// TIA Portal project "DT_PSA_OPCV" (V19)

(* hardware
DEVICE "S7-1500/ET200MP-Station_1"  S7-1500 station
   slot 0: "Profilschiene_0"  Rack  6ES7 590-1***0-0AA0
   slot 1: "PLC_1"  CPU 1516F-3 PN/DP  6ES7 516-3FN02-0AB0  V2.9
      slot 3: "CPU-Display_1"  6ES7591-1BA00-0AA0
      slot 32768: "PROFINET-Schnittstelle_1"  X1
         slot 32769: "Port_1"  X1 P1
         slot 32770: "Port_2"  X1 P2
      slot 33024: "PROFINET-Schnittstelle_2"  X2
         slot 33025: "Port_1"  X2 P1
      slot 33280: "DP-Schnittstelle_1"  X3
      slot 34817: "Virtual CP interface port_1"  Virtual CP interface port  Virtual CP interface port
   slot 2: "DI 16x24VDC HF_1"  DI 16x24VDC HF  6ES7 521-1BH00-0AB0  V2.2
   slot 3: "DQ 8x24VDC/2A HF_1"  DQ 8x24VDC/2A HF  6ES7 522-1BF00-0AB0  V2.2
   slot 4: "F-DI 16x24V DC_1"  F-DI 16x24V DC  6ES7 526-1BH00-0AB0  V1.0
      slot 1: "F-DI 16x24V DC_1"  F-DI 16x24V DC
   slot 5: "F-DQ 8x24V DC/2A PPM_1"  F-DQ 8x24V DC/2A PPM  6ES7 526-2BF00-0AB0  V1.0
      slot 1: "F-DQ 8x24V DC/2A PPM_1"  F-DQ 8x24V DC/2A PPM
DEVICE "HMI_1"  TP700 Comfort
   slot 0: "HMI_1"  TP700 Comfort  6AV2 124-0GC01-0AX0  17.0.0.0
   slot 1: "HMI_RT_1"  TP700 Comfort  6AV2 124-0GC01-0AX0  17.0.0.0
   slot 5: "HMI_1.IE_CP_1"  PROFINET Interface  17.0.0.0
      slot 1: "PROFINET Schnittstelle_1"  PROFINET Interface
         slot 1: "Port_1"  Port
         slot 2: "Port_2"  Port
   slot 7: "HMI_1.MPI/DP_CP_1"  MPI/DP Interface  17.0.0.0
*)

// ===== PLC "PLC_1"  CPU 1516F-3 PN/DP =====
// protected blocks, not shown: "Main_Safety_RTG1", "Main_Safety_RTG1_DB"

VAR_GLOBAL   // PLC tag table "Control Panel"
   "BT2_OpMode" AT %I0.2 : Bool;   // Betriebsart: 1=Automatik / 0=Hand / Operating mode: 1 = Automatic / 0 = Manual
   "BT3_SingleStep" AT %I0.3 : Bool;   // Einzelschritt ausführen / Execute single step
   "BT4_AutoStart" AT %I0.4 : Bool;   // Automatik Ein / Automatic on
   "BT5_AutoStop" AT %I0.5 : Bool;   // Automatik Halt / Automatic stop
   "BT7_Reset" AT %I0.7 : Bool;   // Grundstellung / Home position
   "BT6_Ack" AT %I0.6 : Bool;   // Störung quittieren / Acknowledge fault
   "BT1_ControlLight" AT %Q0.1 : Bool;   // Tasterbeleuchtung "Steuerung läuft" (grün) / Pushbutton illumination: "Control running" (green)
   "BT4_AutoLight" AT %Q0.4 : Bool;   // Tasterbeleuchtung "Automatik läuft" (grün) / Pushbutton illumination: "Automatic running" (green)
   "BT6_ErrFltLight" AT %Q0.6 : Bool;   // Tasterbeleuchtung "Lampe Störung" (rot) / Pushbutton illumination: "Fault indicator" (red)
   "SignalTower_Yellow" AT %Q1.2 : Bool;   // Ampel "Lampe Einrichten aktiv" (gelb) / Signal tower: "Setup active" (yellow)
   "BT1_ControlOnOff" AT %I0.1 : Bool;   // 1 = Steuerung Ein (einrastend) / 1 = Control on (latching)
   "SignalTower_Green" AT %Q1.1 : Bool;   // Ampel "Automatik läuft" (grün) / Signal tower: "Automatic running" (green)
   "SignalTower_Red" AT %Q1.3 : Bool;   // Ampel "Störung" (rot) / Signal tower: "Fault" (red)
   "BT3_SingleStepLight" AT %Q0.3 : Bool;   // Tasterbeleuchtung "Einzelschritt läuft" (grün) / Pushbutton illumination: "Single step running" (green)
   "BT7_HomingLight" AT %Q0.7 : Bool;   // Tasterbeleuchtung „Grundstellungsfahrt läuft“ (grün) / Pushbutton illumination: "Homing in progress" (green)
   "BT5_AutoStopLight" AT %Q0.5 : Bool;   // Tasterbeleuchtung "Automatikstopp läuft" (blau) / Pushbutton illumination: "Automatic stopping" (blue)
   "BT8_ImmediateStop" AT %I1.0 : Bool;   // Sofort Halt / Immediate stop
   "BT8_ImmediateStopLight" AT %Q1.0 : Bool;   // Tasterbeleuchtung "Sofort Halt" (rot) / Pushbutton illumination: "Immediate stop" (red)
   "SignalTower_Blue" AT %Q1.4 : Bool;   // Ampel "Automatik stoppt" (blau) / Signal tower: "Automatic stopping" (blue)
   "q_SS_ESTOP1" AT %Q0.0 : Bool;   // Beleuchtung Not-Aus 1 / Emergency stop 1 illumination
   "q_SS_ESTOP2" AT %Q0.2 : Bool;   // Beleuchtung Not-Aus 2 / Emergency stop 2 illumination
END_VAR

VAR_GLOBAL   // PLC tag table "System"
   "Clock_Byte" AT %MB0 : Byte;
   "Clock_10Hz" AT %M0.0 : Bool;
   "Clock_5Hz" AT %M0.1 : Bool;
   "Clock_2.5Hz" AT %M0.2 : Bool;
   "Clock_2Hz" AT %M0.3 : Bool;
   "Clock_1.25Hz" AT %M0.4 : Bool;
   "Clock_1Hz" AT %M0.5 : Bool;
   "Clock_0.625Hz" AT %M0.6 : Bool;
   "Clock_0.5Hz" AT %M0.7 : Bool;
   "System_Byte" AT %MB1 : Byte;
   "FirstScan" AT %M1.0 : Bool;
   "DiagStatusUpdate" AT %M1.1 : Bool;
   "AlwaysTRUE" AT %M1.2 : Bool;
   "AlwaysFALSE" AT %M1.3 : Bool;
   "Commissioning_True" AT %M2.0 : Bool;
END_VAR

VAR_GLOBAL CONSTANT   // PLC tag table "System"
   "SYS_MACHINE_MAXSTATIONS" : USInt := 10;   // Anzahl Stationen pro Maschine / Number of stations per machine
   "SYS_SQ_MAXSEQUENCES" : USInt := 12;   // Anzahl Schrittketten pro Station / Number of sequences per station
   "SYS_DRIVE_POSITIONS" : USInt := 8;   // Anzahl Positionen pro Servoantrieb / Number of positions per servo drive
   "SYS_MANUALMOVEMENTS" : UInt := 64;   // Maximale Anzahl an Einrichtfunktionen / Maximum number of setup functions
   "SYS_HMI_SETUPMAXROWS" : USInt := 6;   // HMI-Vorgabe: maximale Anzahl der auf der Steuerung verfügbaren Einrichtzeilen / HMI setting: maximum number of setup rows available on the PLC
   "SYS_CYCLETIMES" : Int := 10;   // Anzahl Zykluszeitauswertungen / Number of cycle time evaluations
END_VAR

VAR_GLOBAL   // PLC tag table "FG01"
   "FG01_Y_Gripper_InHome" AT %I101.0 : Bool;   // geöffnet / open
   "FG01_Y_Gripper_InWork" AT %I101.1 : Bool;   // geschlossen / closed
   "FG01_Y_Gripper_WorkPos" AT %Q101.1 : Bool;   // schließen / close
   "FG01_Y_Plattform_InHome" AT %I102.0 : Bool;   // hinten / rear
   "FG01_Y_Plattform_InWork" AT %I102.1 : Bool;   // vorne / front
   "FG01_Y_Plattform_HomePos" AT %Q102.0 : Bool;
   "FG01_Y_Plattform_WorkPos" AT %Q102.1 : Bool;
   "FG01_Y_ReaderWindow_InWork" AT %I103.1 : Bool;
   "FG01_Y_ReaderWindow_WorkPos" AT %Q103.1 : Bool;   // Position zum Lesen des Codes / Code reading position
   "FG01_Y_Gripper_HomePos" AT %Q101.0 : Bool;   // öffnen / open
   "FG01_Y_ReaderWindow_HomePos" AT %Q103.0 : Bool;
   "FG01_Y_Gate_1_InHome" AT %I104.0 : Bool;   // geöffnet / open
   "FG01_Y_Gate_1_InWork" AT %I104.1 : Bool;   // geschlossen / closed
   "FG01_Y_Gate_1_WorkPos" AT %Q104.1 : Bool;   // Schließen / Close
   "FG01_Y_Gate_2_InHome" AT %I105.0 : Bool;   // geöffnet / open
   "FG01_Y_Gate_2_InWork" AT %I105.1 : Bool;   // geschlossen / closed
   "FG01_Y_Gate_2_WorkPos" AT %Q105.1 : Bool;   // Schließen / Close
   "FG01_Y_LaserMark" AT %Q107.0 : Bool;
   "FG01_P_Camera.bEnable" AT %Q108.0 : Bool;
   "FG01_P_Camera.bTrigger" AT %Q108.1 : Bool;
   "FG01_P_Camera.bReady" AT %I108.0 : Bool;
   "FG01_P_Camera.bBusy" AT %I108.1 : Bool;
   "FG01_P_Camera.bResultValid" AT %I108.2 : Bool;
   "FG01_P_Camera.bResultOk" AT %I108.3 : Bool;
END_VAR

VAR_GLOBAL   // PLC tag table "FG02"
   "FG02_P_Camera.bEnable" AT %Q200.0 : Bool;
   "FG02_P_Camera.bTrigger" AT %Q200.1 : Bool;
   "FG02_P_Camera.bReady" AT %I200.0 : Bool;
   "FG02_P_Camera.bBusy" AT %I200.1 : Bool;
   "FG02_P_Camera.bResultValid" AT %I200.2 : Bool;
   "FG02_P_Camera.bResultOk" AT %I200.3 : Bool;
END_VAR

VAR_GLOBAL   // PLC tag table "FG03"
   "FG03_Y_AxisR1_InHome" AT %I301.0 : Bool;
   "FG03_Y_AxisR1_InWork" AT %I301.1 : Bool;
   "FG03_Y_AxisR1_HomePos" AT %Q301.0 : Bool;
   "FG03_Y_AxisR1_WorkPos" AT %Q301.1 : Bool;
   "FG03_Y_AxisX1_InHome" AT %I302.0 : Bool;
   "FG03_Y_AxisX1_InWork" AT %I302.1 : Bool;
   "FG03_Y_AxisX1_HomePos" AT %Q302.0 : Bool;
   "FG03_Y_AxisX1_WorkPos" AT %Q302.1 : Bool;
   "FG03_Y_AxisY1_InHome" AT %I303.0 : Bool;
   "FG03_Y_AxisY1_InWork" AT %I303.1 : Bool;
   "FG03_Y_AxisY1_HomePos" AT %Q303.0 : Bool;
   "FG03_Y_AxisY1_WorkPos" AT %Q303.1 : Bool;
   "FG03_Y_AxisX2_InHome" AT %I304.0 : Bool;
   "FG03_Y_AxisX2_InWork" AT %I304.1 : Bool;
   "FG03_Y_AxisX2_HomePos" AT %Q304.0 : Bool;
   "FG03_Y_AxisX2_WorkPos" AT %Q304.1 : Bool;
   "FG03_Y_AxisY2_InHome" AT %I305.0 : Bool;
   "FG03_Y_AxisY2_InWork" AT %I305.1 : Bool;
   "FG03_Y_AxisY2_HomePos" AT %Q305.0 : Bool;
   "FG03_Y_AxisY2_WorkPos" AT %Q305.1 : Bool;
   "FG03_Y_Gripper1_InHome" AT %I306.0 : Bool;
   "FG03_Y_Gripper1_InWork" AT %I306.1 : Bool;
   "FG03_Y_Gripper1_HomePos" AT %Q306.0 : Bool;
   "FG03_Y_Gripper1_WorkPos" AT %Q306.1 : Bool;
   "FG03_Y_Gripper2_InHome" AT %I307.0 : Bool;
   "FG03_Y_Gripper2_InWork" AT %I307.1 : Bool;
   "FG03_Y_Gripper2_HomePos" AT %Q307.0 : Bool;
   "FG03_Y_Gripper2_WorkPos" AT %Q307.1 : Bool;
END_VAR

VAR_GLOBAL   // PLC tag table "FG04"
   "FG04_Y_AxisZ_InWork" AT %I401.1 : Bool;
   "FG04_Y_AxisZ_WorkPos" AT %Q401.1 : Bool;
   "FG04_Y_AxisZ_HomePos" AT %Q401.0 : Bool;
   "FG04_Y_AxisZ_InHome" AT %I401.0 : Bool;
END_VAR

VAR_GLOBAL   // PLC tag table "FG05"
   "FG05_B_Part" AT %I500.0 : Bool;
   "FG05_Y_AxisR_InHome" AT %I501.0 : Bool;
   "FG05_Y_AxisR_InWork" AT %I501.1 : Bool;
   "FG05_Y_AxisR_HomePos" AT %Q501.0 : Bool;
   "FG05_Y_AxisR_WorkPos" AT %Q501.1 : Bool;
   "FG05_Y_AxisX_InHome" AT %I502.0 : Bool;
   "FG05_Y_AxisX_InWork" AT %I502.1 : Bool;
   "FG05_Y_AxisX_HomePos" AT %Q502.0 : Bool;
   "FG05_Y_AxisX_WorkPos" AT %Q502.1 : Bool;
   "FG05_Y_AxisZ1_InHome" AT %I503.0 : Bool;
   "FG05_Y_AxisZ1_InWork" AT %I503.1 : Bool;
   "FG05_Y_AxisZ1_HomePos" AT %Q503.0 : Bool;
   "FG05_Y_AxisZ1_WorkPos" AT %Q503.1 : Bool;
   "FG05_Y_AxisZ2_InHome" AT %I504.0 : Bool;
   "FG05_Y_AxisZ2_InWork" AT %I504.1 : Bool;
   "FG05_Y_AxisZ2_HomePos" AT %Q504.0 : Bool;
   "FG05_Y_AxisZ2_WorkPos" AT %Q504.1 : Bool;
   "FG05_Y_CapsSourceStopper_InHome" AT %I505.0 : Bool;   // GS = Kappen können vereinzelt werden / GS = Caps can be separated
   "FG05_Y_CapsSourceStopper_WorkPos" AT %Q505.1 : Bool;   // AS = Vereinzelung kann geleert werden (Vereinzelung nicht möglich) / AS = Separator can be emptied (separation not possible)
   "FG05_Y_Gripper_InHome" AT %I506.0 : Bool;
   "FG05_Y_Gripper_InWork" AT %I506.1 : Bool;
   "FG05_Y_Gripper_HomePos" AT %Q506.0 : Bool;
   "FG05_Y_Gripper_WorkPos" AT %Q506.1 : Bool;
   "FG05_Y_CapsSourceStopper_HomePos" AT %Q505.0 : Bool;
   "FG05_M_Bunker" AT %Q507.0 : Bool;   // Sortiertopf ein / Bowl feeder on
   "FG05_M_Conveyor" AT %Q507.1 : Bool;   // Linearförderer ein / Linear conveyor on
   "FG05_P_Camera.bEnable" AT %Q508.0 : Bool;
   "FG05_P_Camera.bTrigger" AT %Q508.1 : Bool;
   "FG05_P_Camera.bReady" AT %I508.0 : Bool;
   "FG05_P_Camera.bBusy" AT %I508.1 : Bool;
   "FG05_P_Camera.bResultValid" AT %I508.2 : Bool;
   "FG05_P_Camera.bResultOk" AT %I508.3 : Bool;
END_VAR

VAR_GLOBAL   // PLC tag table "FG_Transport"
   "FG_TS_Index01_B_Detect" AT %I1003.0 : Bool;   // 1 = erkannt / 1 = Detected
   "FG_TS_Index01_B_Exit" AT %I1003.1 : Bool;   // 1 = erkannt / 1 = Detected
   "FG_TS_Index01_Y_Lift_InHome" AT %I1003.2 : Bool;   // Heber ist unten / Lift is down
   "FG_TS_Index01_Y_Lift_InWork" AT %I1003.3 : Bool;   // Heber ist oben / Lift is up
   "FG_TS_Index01_Y_Lift_HomePos" AT %Q1003.0 : Bool;   // Heber senken / Lower lift
   "FG_TS_Index01_Y_Lift_WorkPos" AT %Q1003.1 : Bool;   // Heber heben / Raise lift
   "FG_TS_Index01_Y_Stopper_InHome" AT %I1003.4 : Bool;   // Stopper geschlossen / Stopper closed
   "FG_TS_Index01_Y_Stopper_WorkPos" AT %Q1003.2 : Bool;   // Stopper öffnen / Open stopper
   "FG_TS_Index02_B_Detect" AT %I1004.0 : Bool;   // 1 = erkannt / 1 = Detected
   "FG_TS_Index02_B_Exit" AT %I1004.1 : Bool;   // 1 = erkannt / 1 = Detected
   "FG_TS_Index02_Y_Lift_InHome" AT %I1004.2 : Bool;   // Heber ist unten / Lift is down
   "FG_TS_Index02_Y_Lift_InWork" AT %I1004.3 : Bool;   // Heber ist oben / Lift is up
   "FG_TS_Index02_Y_Lift_HomePos" AT %Q1004.0 : Bool;   // Heber senken / Lower lift
   "FG_TS_Index02_Y_Lift_WorkPos" AT %Q1004.1 : Bool;   // Heber heben / Raise lift
   "FG_TS_Index02_Y_Stopper_InHome" AT %I1004.4 : Bool;   // Stopper geschlossen / Stopper closed
   "FG_TS_Index02_Y_Stopper_WorkPos" AT %Q1004.2 : Bool;   // Stopper öffnen / Open stopper
   "FG_TS_Index03_B_Detect" AT %I1005.0 : Bool;   // 1 = erkannt / 1 = Detected
   "FG_TS_Index03_B_Exit" AT %I1005.1 : Bool;   // 1 = erkannt / 1 = Detected
   "FG_TS_Index03_Y_Lift_InHome" AT %I1005.2 : Bool;   // Heber ist unten / Lift is down
   "FG_TS_Index03_Y_Lift_InWork" AT %I1005.3 : Bool;   // Heber ist oben / Lift is up
   "FG_TS_Index03_Y_Lift_HomePos" AT %Q1005.0 : Bool;   // Heber senken / Lower lift
   "FG_TS_Index03_Y_Lift_WorkPos" AT %Q1005.1 : Bool;   // Heber heben / Raise lift
   "FG_TS_Index03_Y_Stopper_InHome" AT %I1005.4 : Bool;   // Stopper geschlossen / Stopper closed
   "FG_TS_Index03_Y_Stopper_WorkPos" AT %Q1005.2 : Bool;   // Stopper öffnen / Open stopper
   "FG_TS_Index04_B_Detect" AT %I1006.0 : Bool;   // 1 = erkannt / 1 = Detected
   "FG_TS_Index04_B_Exit" AT %I1006.1 : Bool;   // 1 = erkannt / 1 = Detected
   "FG_TS_Index04_Y_Lift_InHome" AT %I1006.2 : Bool;   // Heber ist unten / Lift is down
   "FG_TS_Index04_Y_Lift_InWork" AT %I1006.3 : Bool;   // Heber ist oben / Lift is up
   "FG_TS_Index04_Y_Lift_HomePos" AT %Q1006.0 : Bool;   // Heber senken / Lower lift
   "FG_TS_Index04_Y_Lift_WorkPos" AT %Q1006.1 : Bool;   // Heber heben / Raise lift
   "FG_TS_Index04_Y_Stopper_InHome" AT %I1006.4 : Bool;   // Stopper geschlossen / Stopper closed
   "FG_TS_Index04_Y_Stopper_WorkPos" AT %Q1006.2 : Bool;   // Stopper öffnen / Open stopper
   "FG_TS_Index05_B_Detect" AT %I1007.0 : Bool;   // 1 = erkannt / 1 = Detected
   "FG_TS_Index05_B_Exit" AT %I1007.1 : Bool;   // 1 = erkannt / 1 = Detected
   "FG_TS_Index05_Y_Lift_InHome" AT %I1007.2 : Bool;   // Heber ist unten / Lift is down
   "FG_TS_Index05_Y_Lift_InWork" AT %I1007.3 : Bool;   // Heber ist oben / Lift is up
   "FG_TS_Index05_Y_Lift_HomePos" AT %Q1007.0 : Bool;   // Heber senken / Lower lift
   "FG_TS_Index05_Y_Lift_WorkPos" AT %Q1007.1 : Bool;   // Heber heben / Raise lift
   "FG_TS_Index05_Y_Stopper_InHome" AT %I1007.4 : Bool;   // Stopper geschlossen / Stopper closed
   "FG_TS_Index05_Y_Stopper_WorkPos" AT %Q1007.2 : Bool;   // Stopper öffnen / Open stopper
   "FG_TS_Stopper01_B_Detect" AT %I1008.0 : Bool;   // 1 = erkannt / 1 = Detected
   "FG_TS_Stopper01_B_Exit" AT %I1008.1 : Bool;   // 1 = erkannt / 1 = Detected
   "FG_TS_Stopper01_Y_Stopper_InHome" AT %I1008.4 : Bool;   // Stopper geschlossen / Stopper closed
   "FG_TS_Stopper01_Y_Stopper_WorkPos" AT %Q1008.2 : Bool;   // Stopper öffnen / Open stopper
   "FG_TS_Stopper02_B_Detect" AT %I1009.0 : Bool;   // 1 = erkannt / 1 = Detected
   "FG_TS_Stopper02_B_Exit" AT %I1009.1 : Bool;   // 1 = erkannt / 1 = Detected
   "FG_TS_Stopper02_Y_Stopper_InHome" AT %I1009.4 : Bool;   // Stopper geschlossen / Stopper closed
   "FG_TS_Stopper02_Y_Stopper_WorkPos" AT %Q1009.2 : Bool;   // Stopper öffnen / Open stopper
   "FG_TS_Stopper03_B_Detect" AT %I1010.0 : Bool;   // 1 = erkannt / 1 = Detected
   "FG_TS_Stopper03_B_Exit" AT %I1010.1 : Bool;   // 1 = erkannt / 1 = Detected
   "FG_TS_Stopper03_Y_Stopper_InHome" AT %I1010.4 : Bool;   // Stopper geschlossen / Stopper closed
   "FG_TS_Stopper03_Y_Stopper_WorkPos" AT %Q1010.2 : Bool;   // Stopper öffnen / Open stopper
   "FG_TS_Stopper04_B_Detect" AT %I1011.0 : Bool;   // 1 = erkannt / 1 = Detected
   "FG_TS_Stopper04_B_Exit" AT %I1011.1 : Bool;   // 1 = erkannt / 1 = Detected
   "FG_TS_Stopper04_Y_Stopper_InHome" AT %I1011.4 : Bool;   // Stopper geschlossen / Stopper closed
   "FG_TS_Stopper04_Y_Stopper_WorkPos" AT %Q1011.2 : Bool;   // Stopper öffnen / Open stopper
   "FG_TS_Lift01_B_Detect" AT %I1012.0 : Bool;   // 1 = erkannt / 1 = Detected
   "FG_TS_Lift01_B_Exit" AT %I1012.1 : Bool;   // 1 = erkannt / 1 = Detected
   "FG_TS_Lift01_Y_Lift_InHome" AT %I1012.2 : Bool;   // Heber ist unten / Lift is down
   "FG_TS_Lift01_Y_Lift_InWork" AT %I1012.3 : Bool;   // Heber ist oben / Lift is up
   "FG_TS_Lift01_Y_Lift_HomePos" AT %Q1012.0 : Bool;   // Heber senken / Lower lift
   "FG_TS_Lift01_Y_Lift_WorkPos" AT %Q1012.1 : Bool;   // Heber heben / Raise lift
   "FG_TS_Lift01_M_Conveyor_Plus" AT %Q1012.2 : Bool;   // Antrieb vorwärts / Drive forwards
   "FG_TS_Lift01_M_Conveyor_Minus" AT %Q1012.3 : Bool;   // Antrieb rückwärts / Drive backwards
   "FG_TS_Lift02_B_Detect" AT %I1013.0 : Bool;   // 1 = erkannt / 1 = Detected
   "FG_TS_Lift02_B_Exit" AT %I1013.1 : Bool;   // 1 = erkannt / 1 = Detected
   "FG_TS_Lift02_Y_Lift_InHome" AT %I1013.2 : Bool;   // Heber ist unten / Lift is down
   "FG_TS_Lift02_Y_Lift_InWork" AT %I1013.3 : Bool;   // Heber ist oben / Lift is up
   "FG_TS_Lift02_Y_Lift_HomePos" AT %Q1013.0 : Bool;   // Heber senken / Lower lift
   "FG_TS_Lift02_Y_Lift_WorkPos" AT %Q1013.1 : Bool;   // Heber heben / Raise lift
   "FG_TS_Lift02_M_Conveyor_Plus" AT %Q1013.2 : Bool;   // Antrieb vorwärts / Drive forwards
   "FG_TS_Lift02_M_Conveyor_Minus" AT %Q1013.3 : Bool;   // Antrieb rückwärts / Drive backwards
   "FG_TS_Transport01_M_Conveyor_Plus" AT %Q1014.0 : Bool;   // Antrieb vorwärts / Drive forwards
   "FG_TS_Transport01_M_Conveyor_Minus" AT %Q1014.1 : Bool;   // Antrieb rückwärts / Drive backwards
   "FG_TS_Transport02_M_Conveyor_Plus" AT %Q1015.0 : Bool;   // Antrieb vorwärts / Drive forwards
   "FG_TS_Transport02_M_Conveyor_Minus" AT %Q1015.1 : Bool;   // Antrieb rückwärts / Drive backwards
END_VAR

VAR_GLOBAL   // PLC tag table "Safety"
   "i_SS_ESTOP1" AT %I50.0 : Bool;
   "i_SS_ESTOP2" AT %I50.1 : Bool;
END_VAR

// folder: Actors/ActorTypes

TYPE "typeActor"
   STRUCT
      setHomePos : Bool;   // Grundstellung ansteuern / Command home position
      setWorkPos : Bool;   // Arbeitsstellung ansteuern / Command working position
      inHomePos : Bool;   // steht in Grundstellung / in home position
      inWorkPos : Bool;   // steht in Arbeitsstellung / in working position
      homeAct : Bool;   // Grundstellung wird angesteuert / Home position commanded
      workAct : Bool;   // Arbeitsstellung wird angesteuert / Working position commanded
      homeIsInterlocked : Bool;   // 1 = Grundstellung ist gesperrt / 1 = Home position movement inhibited
      workIsInterlocked : Bool;   // 1 = Arbeitsstellung ist gesperrt / 1 = Working position movement inhibited
   END_STRUCT;
END_TYPE

TYPE "typeActor_2Out0In"
   STRUCT
      setHomePos : Bool;   // Grundstellung ansteuern / Command home position
      setWorkPos : Bool;   // Arbeitsstellung ansteuern / Command working position
      homeAct : Bool;   // Grundstellung wird angesteuert / Home position commanded
      workAct : Bool;   // Arbeitsstellung wird angesteuert / Working position commanded
      homeIsInterlocked : Bool;   // 1 = Grundstellung ist gesperrt / 1 = Home position movement inhibited
      workIsInterlocked : Bool;   // 1 = Arbeitsstellung ist gesperrt / 1 = Working position movement inhibited
      setError : Bool;   // in Störung setzen / Set fault state
      inError : Bool;   // Störung vorhanden / Fault present
   END_STRUCT;
END_TYPE

TYPE "typeActor_2Out2In"
   STRUCT
      setHomePos : Bool;   // Grundstellung ansteuern / Command home position
      setWorkPos : Bool;   // Arbeitsstellung ansteuern / Command working position
      inHomePos : Bool;   // steht in Grundstellung / in home position
      inWorkPos : Bool;   // steht in Arbeitsstellung / in working position
      homeAct : Bool;   // Grundstellung wird angesteuert / Home position commanded
      workAct : Bool;   // Arbeitsstellung wird angesteuert / Working position commanded
      homeIsInterlocked : Bool;   // 1 = Grundstellung ist gesperrt / 1 = Home position movement inhibited
      workIsInterlocked : Bool;   // 1 = Arbeitsstellung ist gesperrt / 1 = Working position movement inhibited
      setError : Bool;   // in Störung setzen / Set fault state
      inError : Bool;   // Störung vorhanden / Fault present
   END_STRUCT;
END_TYPE

TYPE "typeActor_1Out0In"
   STRUCT
      setWorkPos : Bool;   // Arbeitsstellung ansteuern / Command working position
      workAct : Bool;   // Arbeitsstellung wird angesteuert / Working position commanded
      workIsInterlocked : Bool;   // 1 = Arbeitsstellung ist gesperrt / 1 = Working position movement inhibited
      setError : Bool;   // in Störung setzen / Set fault state
      inError : Bool;   // Störung vorhanden / Fault present
   END_STRUCT;
END_TYPE

TYPE "typeActor_1Out2In"
   STRUCT
      setWorkPos : Bool;   // Arbeitsstellung ansteuern / Command working position
      inHomePos : Bool;   // steht in Grundstellung / in home position
      inWorkPos : Bool;   // steht in Arbeitsstellung / in working position
      workAct : Bool;   // Arbeitsstellung wird angesteuert / Working position commanded
      workIsInterlocked : Bool;   // 1 = Arbeitsstellung ist gesperrt / 1 = Working position movement inhibited
      setError : Bool;   // in Störung setzen / Set fault state
      inError : Bool;   // Störung vorhanden / Fault present
   END_STRUCT;
END_TYPE

TYPE "typeActor_2Out1In"
   STRUCT
      setHomePos : Bool;   // Grundstellung ansteuern / Command home position
      setWorkPos : Bool;   // Arbeitsstellung ansteuern / Command working position
      inHomePos : Bool;   // steht in Grundstellung / in home position
      inWorkPos : Bool;   // steht in Arbeitsstellung / in working position
      homeAct : Bool;   // Grundstellung wird angesteuert / Home position commanded
      workAct : Bool;   // Arbeitsstellung wird angesteuert / Working position commanded
      homeIsInterlocked : Bool;   // 1 = Grundstellung ist gesperrt / 1 = Home position movement inhibited
      workIsInterlocked : Bool;   // 1 = Arbeitsstellung ist gesperrt / 1 = Working position movement inhibited
      setError : Bool;   // in Störung setzen / Set fault state
      inError : Bool;   // Störung vorhanden / Fault present
   END_STRUCT;
END_TYPE

TYPE "typeActor_1Out1In"
   STRUCT
      setWorkPos : Bool;   // Arbeitsstellung ansteuern / Command working position
      inHomePos : Bool;   // steht in Grundstellung / in home position
      inWorkPos : Bool;   // steht in Arbeitsstellung / in working position
      workAct : Bool;   // Arbeitsstellung wird angesteuert / Working position commanded
      workIsInterlocked : Bool;   // 1 = Arbeitsstellung ist gesperrt / 1 = Working position movement inhibited
      setError : Bool;   // in Störung setzen / Set fault state
      inError : Bool;   // Störung vorhanden / Fault present
   END_STRUCT;
END_TYPE

TYPE "typeActor_1Out_SimpleCamera"
   STRUCT
      setTrigger : Bool;   // Kamera auslösen / Trigger camera
      isReady : Bool;   // ist bereit / ready
      isBusy : Bool;   // ist aktiv / active
      resultOk : Bool;   // Ergebnis ist IO / Result OK
      resultNok : Bool;   // Ergebnis ist NIO / Result NOK
      triggerAct : Bool;   // Trigger wird angesteuert / Trigger commanded
      workIsInterlocked : Bool;   // Triggern ist gesperrt / Triggering inhibited
      setError : Bool;   // in Störung setzen / Set fault state
      inError : Bool;   // Störung vorhanden / Fault present
   END_STRUCT;
END_TYPE

// folder: Actors/Drives

TYPE "typeDriveData"
   STRUCT
      position : Array[1.."SYS_DRIVE_POSITIONS"] of Real;   // Positionsvorgabe / Position setpoint
      speed : Array[1.."SYS_DRIVE_POSITIONS"] of Real;   // Geschwindigkeitsvorgabe / Speed setpoint
   END_STRUCT;
   // // position[1] : Grundstellung (reserviert) / Home position (reserved)
END_TYPE

TYPE "typeDriveControl"
   STRUCT
      moveToPos : Array[1.."SYS_DRIVE_POSITIONS"] of Bool;   // Fahrbefehl ausführen / Execute motion command
      jog : Struct   // Handbetrieb / Manual operation
         pos : Bool;   // Tippen positiv / Jog positive
         neg : Bool;   // Tippen negativ / Jog negative
         "step" : Real;   // Tippschrittweite / Jog increment
         speed : Real;   // Tippgeschwindigkeit / Jog speed
      END_STRUCT;
   END_STRUCT;
END_TYPE

TYPE "typeDriveStatus"
   STRUCT
      ready : Bool;   // Bereit / Ready
      error : Bool;   // Störung / Fault
      posReached : Bool;   // Positionsvorgabe erreicht / Position setpoint reached
      actualPosition : Real;   // Ist-Position / Actual position
      actualSpeed : Real;   // Ist-Geschwindigkeit / Actual speed
      interlockMin : Bool;   // 1 = Fahrtrichtung zur Endposition min gesperrt / 1 = Movement towards minimum end position inhibited
      interlockMax : Bool;   // 1 = Fahrtrichtung zur Endposition max gesperrt / 1 = Movement towards maximum end position inhibited
      endPosMin : Bool;   // Endposition min erreicht / Minimum end position reached
      endPosMax : Bool;   // Endposition max erreicht / Maximum end position reached
      inHomePos : Bool;   // steht in Grundstellung / in home position
   END_STRUCT;
END_TYPE

TYPE "typeDriveConverter"
   STRUCT
      actualPosition : Real;   // Ist-Position (Antriebseinheit) / Actual position (drive units)
      actualSpeed : Real;   // Ist-Geschwindigkeit (Antriebseinheit) / Actual speed (drive units)
      setPosition : Real;   // Sollposition (Antriebseinheit) / Target position (drive units)
      setSpeed : Real;   // Sollgeschwindigkeit (Antriebseinheit) / Target speed (drive units)
      minPosDrive : Real;   // Minimale Positionierung (Antriebseinheit) / Minimum positioning value (drive units)
      maxPosDrive : Real;   // Maximale Positionierung (Antriebseinheit) / Maximum positioning value (drive units)
      maxSpeedDrive : Real;   // Maximale Geschwindigkeit (Antriebseinheit) / Maximum speed (drive units)
      posOffset : Real;   // Offset für Positionsfensterfreigabe (Antriebseinheit) / Offset for position window enable (drive units)
      ready : Bool;   // Umrichter Bereit / Converter ready
      error : Bool;   // Umrichter Störung / Converter fault
      posReached : Bool;   // Position erreicht / Position reached
      releaseMotion : Bool;   // Bewegungsfreigabe / Movement enable
   END_STRUCT;
END_TYPE

// folder: HMI/Errors_Messages

TYPE "typePlcErrors"
   STRUCT
      errorNo : Array[1..64] of Bool;
   END_STRUCT;
END_TYPE

TYPE "typeHmiErrMsg"
   STRUCT
      message : Array[1..2] of Word;   // Meldung auslösen / Trigger message
      alarmAckPlc : Array[1..8] of Word;   // Fehler auslösen und Quittierung über SPS / Trigger fault and acknowledge via PLC
      ackHmi : Array[1..4] of Word;   // Quittierung über HMI / Acknowledge via HMI
   END_STRUCT;
END_TYPE

TYPE "typePlcErrMsg"
   STRUCT
      messages : "typePlcMessages";
      alarms : "typePlcErrors";
   END_STRUCT;
END_TYPE

TYPE "typePlcMessages"
   STRUCT
      msgNo : Array[1..32] of Bool;
   END_STRUCT;
END_TYPE

// folder: HMI/ManualMovement

TYPE "typeHmiManualMove"
   STRUCT
      move : "typeManualMove";   // Bewegung / Movement
      movementNo : USInt;   // Nummer der Bewegungsfunktion / Movement function number
      textlistFunctionName : UInt;   // Funktionsname: Wert für Textliste / Function name: text list value
      textlistFunctionExecuteLeft : UInt;   // Bewegung Links: Wert für Textliste / Left movement: text list value
      textlistFunctionFinalPosLeft : UInt;   // Endposition Links: Wert für Textliste / Left end position: text list value
      textlistFunctionExecuteRight : UInt;   // Bewegung Rechts: Wert für Textliste / Right movement: text list value
      textlistFunctionFinalPosRight : UInt;   // Endposition Rechts: Wert für Textliste / Right end position: text list value
   END_STRUCT;
END_TYPE

TYPE "typeHmiManualMovement"
   STRUCT
      selection : Struct
         station : USInt;   // Angewählte Station / Selected station
         page : USInt;   // Aktuelle Seite / Current page
         ofMaxPages : USInt;   // von insgesamt verfügbaren Seiten / of total pages
         nextPage : Bool;   // Schaltfläche: Nächste Seite / Button: Next page
         previousPage : Bool;   // Schaltfläche: Vorherige Seite / Button: Previous page
         showSymbols : Bool;   // Schaltfläche: Zeige symbolische Ansicht / Button: Show symbolic view
      END_STRUCT;
      rows : Array[1.."SYS_HMI_SETUPMAXROWS"] of "typeHmiManualMove";
   END_STRUCT;
END_TYPE

// folder: Machine

TYPE "typeMachine"
   STRUCT
      EStopOk : Bool;   // Not-Aus-Kreis ist geschlossen / Emergency stop circuit closed
      RunUpIsActive : Bool;   // Maschinenanlauf aktiv (Hauptluft einschalten, externe Geräte und Hardware hochfahren) / Machine startup active (switch on main air, start external devices and hardware)
      controlOn : Bool;   // Maschinensteuerung ist eingeschaltet / Machine control switched on
      automaticMode : Bool;   // Betriebsart Automatik ist aktiv / Automatic operating mode active
      automaticIsRunning : Bool;   // Automatik (bzw. ReleaseCycle) läuft in mindestens einer Station / Automatic operation (or ReleaseCycle) running in at least one station
      automaticStart : Bool;   // Automatikstart auslösen / Initiate automatic start
      automaticStops : Bool;   // Automatik stoppt / Automatic stopping
      singleStepPulse : Bool;   // Einzelschritt / Single step
      immediateStop : Bool;   // Sofort Halt der Stationen auslösen / Initiate immediate stop of stations
      acknowledge : Bool;   // Quittierung / Acknowledgement
      reset : Bool;   // Neustart/Grundstellung auslösen / Initiate restart/homing
      isInHoldReached : Bool;   // Alle Stationen haben den Haltepunkt erreicht / All stations have reached the stop point
      isInError : Bool;   // Störung vorhanden / Fault present
      isHoming : Bool;   // Maschinengrundstellungsfahrt wird ausgeführt / Machine homing in progress
      isInHome : Bool;   // Alle Stationen sind in Grundstellung / All stations in home position
   END_STRUCT;
END_TYPE

TYPE "typeStation"
   STRUCT
      xExists : Bool := false;   // true = Station existiert / false = Platzhalter / true = Station exists / false = Placeholder
      usiState : USInt;   // 0 = Bearbeitung, 1 = Störung, 2 = Leerlauf, 3 = Nicht in Produktion, 4 = Warten auf Bediener, 5 = Blockiert, 6 = Materialmangel / 0 = Processing, 1 = Fault, 2 = Idle, 3 = Not in production, 4 = Waiting for operator, 5 = Blocked, 6 = Starved
      udtCycleTime : "typeCycleTime";
      udtSignals : "typeStationSignals";
      udtStepSeqs : "typeStepSequences";
   END_STRUCT;
END_TYPE

TYPE "typeStations"
   STRUCT
      station : Array[1.."SYS_MACHINE_MAXSTATIONS"] of "typeStation";
   END_STRUCT;
END_TYPE

TYPE "typeStepSequence"
   STRUCT
      exists : Bool;   // Schrittkette verfügbar / Sequence available
      start : Bool;   // Start Schrittkette / Start sequence
      running : Bool;   // Schrittkette läuft / Sequence running
      done : Bool;   // Schrittkette ist fertig / Sequence complete
      error : Bool;   // Störung vorhanden / Fault present
      init : Bool;   // Initialschritt aktiv / Initial step active
      inHome : Bool;   // Steht in Grundstellung / In home position
      isWaiting : Bool;   // Steht im Warteschritt / Waiting step active
      inHoming : Bool;   // Grundstellungsfahrt aktiv / Homing active
      jogDone : Bool;   // Halbautomatische Weiterschaltung abgeschlossen / Semi-automatic step advance complete
   END_STRUCT;
END_TYPE

TYPE "typeStepSequences"
   STRUCT
      stepSeq : Array[1.."SYS_SQ_MAXSEQUENCES"] of "typeStepSequence";   // Schrittkette / Sequence
   END_STRUCT;
END_TYPE

TYPE "typeMachineSafety"
   STRUCT
      EStopReq : Bool;   // Not-Aus-Kreis Quittierung erforderlich / Emergency stop circuit acknowledgement required
      EStopOk : Bool;   // Not-Aus-Kreis ok / Emergency stop circuit OK
      RunUp : Bool;   // Hochlaufphase (Starte Belüftung der Hauptventilstation) / Startup phase (start pressurising main valve manifold)
      RunUpIsOk : Bool;   // Sicherheitssteuerung ist hochgefahren (Hauptluftversorgung vorhanden, etc) / Safety control started up (main air supply available, etc.)
      Error : Bool;   // Fehler in der Sicherheitssteuerung / Safety control fault
   END_STRUCT;
END_TYPE

TYPE "typeStationSignals"
   STRUCT
      controlOn : Bool;   // Steuerung eingeschaltet / Control switched on
      automaticMode : Bool;   // Automatikmodus angewählt / Automatic mode selected
      modeSetup : Bool;   // Handmodus angewählt / Manual mode selected
      modeAuto : Bool;   // Betriebsart: Automatik aktiv / Operating mode: Automatic active
      modeTap : Bool;   // Betriebsart: Einzelschritt aktiv / Operating mode: Single step active
      releaseCycle : Bool;   // Bearbeitungsfreigabe / Processing enable
      releaseNextJog : Bool;   // Freigabe Weiterschaltung (Zünd-Impuls für Schrittketten) / Step advance enable (trigger pulse for sequences)
      resetCycle : Bool;   // Ablauf neu starten / Restart sequence
      setupActive : Bool;   // Handmodus/Einrichten aktiv (mindestens 1 Aktor ist in Hand bewegt worden) / Manual/setup mode active (at least one actuator moved manually)
      ack : Bool;   // Quittieren / Acknowledge
      singlePulse : Bool;   // Einzelschritt auslösen / Trigger single step
      safetyIsClosed : Bool;   // Sicherheitskreis ist geschlossen / Safety circuit closed
      safetyIsOk : Bool;   // Sicherheitskreis ist geschlossen und verriegelt / Safety circuit closed and locked
      isInAutoStoping : Bool;   // Automatikstopp/Zyklusende angewählt / Automatic stop / end of cycle selected
      isInHoldReached : Bool;   // Haltepunkt wurde erreicht (z. B. Freigabe zum Öffnen des Sicherheitskreises) / Stop point reached (e.g. permission to open safety circuit)
      isStopped : Bool;   // Automatikabläufe/Graphen sind angehalten / Automatic sequences / GRAPH sequences stopped
      isHoming : Bool;   // Grundstellungsablauf aktiv / Homing sequence active
      isInHome : Bool;   // steht in Grundstellung / in home position
      isInError : Bool;   // Störung vorhanden / Fault present
      actorError : Bool;   // Mindestens ein Stationsaktor hat eine Störung (wird in Aktor-Bausteinen gesetzt) / At least one station actuator has a fault (set in actuator blocks)
      internError : Bool;   // Interner Fehler im Framework vorhanden / Internal framework fault present
   END_STRUCT;
END_TYPE

// folder: Machine/Diag

TYPE "typeCycleTime2"
   STRUCT
      xExists : Bool;   // Zykluszeitauswertung vorhanden / Cycle time evaluation available
      xBottleneck : Bool;   // Bei "true" wird dieser Messbereich zur Diagnose der Engpassstelle ausgewertet / If "true", this measurement area is evaluated for bottleneck diagnosis
      xNewCycle : Bool;   // Ein neuer Messwert liegt vor / New measured value available
      udtHmi : "typeCycleTimeHmi";
      stCurrentCycle : Struct   // Aktueller Zyklus / Current cycle
         tActive : Time;   // Aktive Zeit / Active time
         tInHold : Time;   // Angehaltene Zeit / Stopped time
         tOverall : Time;   // Gesamt / Total
      END_STRUCT;
      stLastCycle : Struct   // Letzter Zyklus / Last cycle
         tActive : Time;   // Aktive Zeit / Active time
         tInHold : Time;   // Angehaltene Zeit / Stopped time
         tOverall : Time;   // Gesamt / Total
      END_STRUCT;
   END_STRUCT;
END_TYPE

TYPE "typeCycleTimes2"
   STRUCT
      cycleTime : Array[1.."SYS_CYCLETIMES"] of "typeCycleTime2";
   END_STRUCT;
END_TYPE

TYPE "typeCycleTimeHmi"
   STRUCT
      rSetpointSeconds : Real := 0.0;   // Sollzeit in Sekunden; Werte kleiner oder gleich 0 deaktivieren die Prüfung / Target time in seconds; values less than or equal to 0 disable the check
      rActiveTimeSeconds : Real;   // Letzte abgeschlossene aktive Zykluszeit in Sekunden / Last completed active cycle time in seconds
      xExceeded : Bool;   // TRUE: Letzte aktive Zykluszeit überschreitet die Sollzeit / TRUE: Last active cycle time exceeds target time
   END_STRUCT;
END_TYPE

TYPE "typeCycleTime"
   STRUCT
      xExists : Bool;   // Zykluszeitauswertung vorhanden / Cycle time evaluation available
      xBottleneck : Bool;   // Bei "true" wird dieser Messbereich zur Diagnose der Engpassstelle ausgewertet / If "true", this measurement area is evaluated for bottleneck diagnosis
      xNewCycle : Bool;   // Ein neuer Messwert liegt vor / New measured value available
      udtHmi : "typeCycleTimeHmi";
      stCurrentCycle : Struct   // Aktueller Zyklus / Current cycle
         tState : Array[0..6] of Time;   // Aktive Zeiten in ms je Stationszustand / Active times in ms per station state
         tOverall : Time;   // Gesamtzeit in ms / Total time in ms
      END_STRUCT;
      stLastCycle : Struct   // Letzter Zyklus / Last cycle
         tState : Array[0..6] of Time;   // Aktive Zeiten in ms je Stationszustand / Active times in ms per station state
         tOverall : Time;   // Gesamtzeit in ms / Total time in ms
      END_STRUCT;
   END_STRUCT;
   // // stCurrentCycle.tState[0] : BEARBEITUNG / PROCESSING
   // // stCurrentCycle.tState[1] : STÖRUNG / FAULT
   // // stCurrentCycle.tState[2] : LEERLAUF / IDLE
   // // stCurrentCycle.tState[3] : NICHT IN PRODUKTION / NOT IN PRODUCTION
   // // stCurrentCycle.tState[4] : WARTEN AUF BEDIENER / WAITING FOR OPERATOR
   // // stCurrentCycle.tState[5] : BLOCKIERT / BLOCKED
   // // stCurrentCycle.tState[6] : MATERIALMANGEL / STARVED
   // // stLastCycle.tState[0] : BEARBEITUNG / PROCESSING
   // // stLastCycle.tState[1] : STÖRUNG / FAULT
   // // stLastCycle.tState[2] : LEERLAUF / IDLE
   // // stLastCycle.tState[3] : NICHT IN PRODUKTION / NOT IN PRODUCTION
   // // stLastCycle.tState[4] : WARTEN AUF BEDIENER / WAITING FOR OPERATOR
   // // stLastCycle.tState[5] : BLOCKIERT / BLOCKED
   // // stLastCycle.tState[6] : MATERIALMANGEL / STARVED
END_TYPE

// folder: Machine/ManualMovement

TYPE "typeManualMove"
   STRUCT
      control : "typeManualMoveControl";   // Steuerung / Control
      attributes : "typeManualMoveAttributes";   // Eigenschaften / Properties
   END_STRUCT;
END_TYPE

TYPE "typeManualMoveSetup"
   STRUCT
      initialisation : Struct   // Für den Initialisierungsdurchlauf notwendig / Required for initialisation pass
         execute : Bool;   // Initialisierung der Bewegungsfunktionen ausführen / Execute movement function initialisation
         isActive : Bool;   // Initialisierung läuft / Initialisation in progress
         isDone : Bool;   // Initialisierung abgeschlossen / Initialisation complete
         error : Bool;   // Initialisierung fehlerhaft / Initialisation failed
         currentStationNo : USInt;   // Hilfsspeicher für die Station / Temporary storage for station
         currentMoveNo : USInt;   // Hilfsspeicher für die Bewegungsnummer innerhalb der Station / Temporary storage for movement number within station
         moveNo : USInt;   // Hilfsspeicher für die Bewegungsnummer (maximale Anzahl Stationen wenn initialisiert) / Temporary movement number storage (maximum station count when initialised)
      END_STRUCT;
   END_STRUCT;
END_TYPE

TYPE "typeManualMovements"
   STRUCT
      setup : "typeManualMoveSetup";
      movements : Array[0.."SYS_MANUALMOVEMENTS"] of "typeManualMove";
   END_STRUCT;
   // // movements[0] : Nicht verwendbar / Not usable
END_TYPE

TYPE "typeManualMoveControl"
   STRUCT
      moveHomePos : Bool;   // Grundstellung ansteuern / Command home position
      moveWorkPos : Bool;   // Arbeitsstellung ansteuern / Command working position
      inHomePos : Bool;   // steht in Grundstellung / in home position
      inWorkPos : Bool;   // steht in Arbeitsstellung / in working position
      homeAct : Bool;   // Grundstellung wird angesteuert / Home position commanded
      workAct : Bool;   // Arbeitsstellung wird angesteuert / Working position commanded
      homeIsInterlocked : Bool;   // 1 = Grundstellung ist gesperrt / 1 = Home position movement inhibited
      workIsInterlocked : Bool;   // 1 = Arbeitsstellung ist gesperrt / 1 = Working position movement inhibited
      value : Real;   // Dezimalanzeige / Decimal display
   END_STRUCT;
END_TYPE

TYPE "typeManualMoveAttributes"
   STRUCT
      initialised : Bool;   // Ist initialisiert / Initialised
      showValue : Bool;   // Zeige Dezimalanzeige / Show decimal display
      showName : Bool;   // Zeige Benennung der Einrichtzeile / Show setup row label
      showRecRight : Bool;   // Rechteck rechts anzeigen / Show right rectangle
      showRecLeft : Bool;   // Rechteck links anzeigen / Show left rectangle
      isExecutableRight : Bool;   // Ist ausführbar rechte Seite / Right side executable
      isExecutableLeft : Bool;   // Ist ausführbar linke Seite / Left side executable
      hasEndPositionRight : Bool;   // Zeige Endposition rechte Seite / Display right end position
      hasEndPositionLeft : Bool;   // Zeige Endposition linke Seite / Display left end position
      stationNo : USInt;   // Zugehörige Stationsnummer / Associated station number
      movementNo : USInt;   // Zugehörige Bewegungsnummer innerhalb der Station / Associated movement number within station
   END_STRUCT;
END_TYPE

// folder: 0.Safety - Password:0000

DATA_BLOCK "SafetySignals"   // DB3
{ S7_Optimized_Access := 'TRUE' }
VERSION : 0.1
   VAR
      xEstop1_Ok : Bool;
      xEstop2_Ok : Bool;
      xEstop1_Ack_Req : Bool;
      xEstop2_Ack_Req : Bool;
   END_VAR
BEGIN
END_DATA_BLOCK

// folder: 1. HMI/TP700_HMI_1

DATA_BLOCK "InstHmiManualMovementController"   // DB1003
{ S7_Optimized_Access := 'TRUE' }
VERSION : 0.1
// stored: InstanceOfName HmiManualMovementController
"HmiManualMovementController"
BEGIN
END_DATA_BLOCK

DATA_BLOCK "HmiManualMovement"   // DB1004
{ S7_Optimized_Access := 'TRUE' }
VERSION : 0.1
BEGIN
END_DATA_BLOCK

// folder: 2. Machine

DATA_BLOCK "InstMachine"   // DB1000
{ S7_Optimized_Access := 'TRUE' }
VERSION : 0.1
// stored: InstanceOfName MachineControl
"MachineControl"
BEGIN
END_DATA_BLOCK

DATA_BLOCK "Machine"   // DB1001
{ S7_Optimized_Access := 'TRUE' }
VERSION : 0.1
   VAR
      safety : "typeMachineSafety";
      machine : "typeMachine";
      stations : "typeStations";
   END_VAR
BEGIN
   // stations.station[1] : FG01
   // stations.station[2] : FG02
   // stations.station[3] : FG03
   // stations.station[4] : FG04
   // stations.station[5] : FG05
   // stations.station[6] : Reserve / Spare
   // stations.station[7] : Reserve / Spare
   // stations.station[8] : Reserve / Spare
   // stations.station[9] : Reserve / Spare
   // stations.station[10] : Transport
   // stations.station[10].udtStepSeqs.stepSeq[1] : Stopper01
   // stations.station[10].udtStepSeqs.stepSeq[2] : Stopper02
   // stations.station[10].udtStepSeqs.stepSeq[3] : Lift01
   // stations.station[10].udtStepSeqs.stepSeq[4] : Stopper03
   // stations.station[10].udtStepSeqs.stepSeq[5] : Index01
   // stations.station[10].udtStepSeqs.stepSeq[6] : Index02
   // stations.station[10].udtStepSeqs.stepSeq[7] : Index03
   // stations.station[10].udtStepSeqs.stepSeq[8] : Index04
   // stations.station[10].udtStepSeqs.stepSeq[9] : Index05
   // stations.station[10].udtStepSeqs.stepSeq[10] : Stopper04
   // stations.station[10].udtStepSeqs.stepSeq[11] : Lift 2
END_DATA_BLOCK

DATA_BLOCK "MachineGlobals"   // DB1002
{ S7_Optimized_Access := 'TRUE' }
VERSION : 0.1
   VAR
      emptying : Bool;   // Maschine leerfahren / Empty machine
   END_VAR
BEGIN
END_DATA_BLOCK

DATA_BLOCK "ManualMovements"   // DB1005
{ S7_Optimized_Access := 'TRUE' }
VERSION : 0.1
BEGIN
END_DATA_BLOCK

// folder: 2. Machine/00_Alarms and Messages

DATA_BLOCK "Alarmserver"   // DB2
{ S7_Optimized_Access := 'TRUE' }
VERSION : 0.1
   VAR
      plc : Struct   // Meldungsspeicher für SPS / Message memory for PLC
         machine : "typePlcErrMsg";
         fg_1 : "typePlcErrMsg";
         fg_2 : "typePlcErrMsg";
         fg_3 : "typePlcErrMsg";
         fg_4 : "typePlcErrMsg";
         fg_5 : "typePlcErrMsg";
         fg_transport : "typePlcErrMsg";
      END_STRUCT;
      hmi : Struct   // Meldungsspeicher für HMI / Message memory for HMI
         machine : "typeHmiErrMsg";
         fg_1 : "typeHmiErrMsg";
         fg_2 : "typeHmiErrMsg";
         fg_3 : "typeHmiErrMsg";
         fg_4 : "typeHmiErrMsg";
         fg_5 : "typeHmiErrMsg";
         fg_transport : "typeHmiErrMsg";
      END_STRUCT;
   END_VAR
BEGIN
END_DATA_BLOCK

// folder: 2. Machine/01_FG01

DATA_BLOCK "InstFG01Control"   // DB1100
{ S7_Optimized_Access := 'TRUE' }
VERSION : 0.1
// stored: InstanceOfName FG01Control
"FG01Control"
BEGIN
END_DATA_BLOCK

DATA_BLOCK "FG01Parameter"   // DB1101
{ S7_Optimized_Access := 'TRUE' }
VERSION : 0.1
BEGIN
END_DATA_BLOCK

DATA_BLOCK "FG01Globals"   // DB1102
{ S7_Optimized_Access := 'TRUE' }
VERSION : 0.1
   VAR
      laserOn : Bool := true;   // Laser einschalten / Switch on laser
      SQ1 : Struct
         readyForIndex : Bool;   // Freigabe für den Indexer zum Anheben / Indexer raising enable
         isinHome : Bool;   // Grundstellung vorhanden / Home position reached
      END_STRUCT;
   END_VAR
BEGIN
END_DATA_BLOCK

DATA_BLOCK "FG01Actors"   // DB1103
{ S7_Optimized_Access := 'TRUE' }
VERSION : 0.1
   VAR
      Gripper : "typeActor_2Out2In";   // Greifer / Gripper
      Plattform : "typeActor_2Out2In";   // Laserplattform / Laser platform
      ReaderWindow : "typeActor_2Out1In";   // Laserplattform / Laser platform
      Lasermarker : "typeActor_1Out0In";   // Lasermarkierer / Laser marker
      Gate_1 : "typeActor_1Out2In";   // Seitentor 1 / Side gate 1
      Gate_2 : "typeActor_1Out2In";   // Seitentor 2 / Side gate 2
      Camera : "typeActor_1Out_SimpleCamera";
   END_VAR
BEGIN
END_DATA_BLOCK

// folder: 2. Machine/01_FG01/Stepsequences

DATA_BLOCK "InstSq_1.1"   // DB1111
{ S7_Optimized_Access := 'TRUE' }
VERSION : 0.1
// stored: InstanceOfName Sq_1.1
"Sq_1.1"
BEGIN
END_DATA_BLOCK

// folder: 2. Machine/02_FG02

DATA_BLOCK "InstFG02Control"   // DB1200
{ S7_Optimized_Access := 'TRUE' }
VERSION : 0.1
// stored: InstanceOfName FG02Control
"FG02Control"
BEGIN
END_DATA_BLOCK

DATA_BLOCK "FG02Globals"   // DB1202
{ S7_Optimized_Access := 'TRUE' }
VERSION : 0.1
   VAR
      SQ1 : Struct
         readyForIndex : Bool;   // Freigabe für den Indexer zum Anheben / Indexer raising enable
         isInHome : Bool;   // Grundstellung vorhanden / Home position reached
      END_STRUCT;
   END_VAR
BEGIN
END_DATA_BLOCK

DATA_BLOCK "FG02Actors"   // DB1203
{ S7_Optimized_Access := 'TRUE' }
VERSION : 0.1
   VAR
      P_Camera : "typeActor_1Out_SimpleCamera";
   END_VAR
BEGIN
END_DATA_BLOCK

// folder: 2. Machine/02_FG02/Stepsequences

DATA_BLOCK "InstSq_2.1"   // DB1211
{ S7_Optimized_Access := 'TRUE' }
VERSION : 0.1
// stored: InstanceOfName Sq_2.1
"Sq_2.1"
BEGIN
END_DATA_BLOCK

// folder: 2. Machine/03_FG03

DATA_BLOCK "InstFG03Control"   // DB1300
{ S7_Optimized_Access := 'TRUE' }
VERSION : 0.1
// stored: InstanceOfName FG03Control
"FG03Control"
BEGIN
END_DATA_BLOCK

DATA_BLOCK "FG03Globals"   // DB1302
{ S7_Optimized_Access := 'TRUE' }
VERSION : 0.1
   VAR
      SQ1 : Struct
         readyForIndex : Bool;   // Freigabe für den Indexer zum Anheben / Indexer raising enable
         isInHome : Bool;   // Grundstellung vorhanden / Home position reached
      END_STRUCT;
   END_VAR
BEGIN
END_DATA_BLOCK

DATA_BLOCK "FG03Actors"   // DB1303
{ S7_Optimized_Access := 'TRUE' }
VERSION : 0.1
   VAR
      AxisR1 : "typeActor_2Out2In";
      AxisX1 : "typeActor_2Out2In";
      AxisY1 : "typeActor_2Out2In";
      AxisX2 : "typeActor_2Out2In";
      AxisY2 : "typeActor_2Out2In";
      Gripper1 : "typeActor_2Out2In";
      Gripper2 : "typeActor_2Out2In";
   END_VAR
BEGIN
END_DATA_BLOCK

// folder: 2. Machine/03_FG03/Stepsequences

DATA_BLOCK "InstSq_3.1"   // DB1311
{ S7_Optimized_Access := 'TRUE' }
VERSION : 0.1
// stored: InstanceOfName Sq_3.1
"Sq_3.1"
BEGIN
END_DATA_BLOCK

// folder: 2. Machine/04_FG04

DATA_BLOCK "InstFG04Control"   // DB1400
{ S7_Optimized_Access := 'TRUE' }
VERSION : 0.1
// stored: InstanceOfName FG04Control
"FG04Control"
BEGIN
END_DATA_BLOCK

DATA_BLOCK "FG04Globals"   // DB1402
{ S7_Optimized_Access := 'TRUE' }
VERSION : 0.1
   VAR
      SQ1 : Struct
         readyForIndex : Bool;   // Freigabe für den Indexer zum Anheben / Indexer raising enable
         isInHome : Bool;   // Grundstellung vorhanden / Home position reached
      END_STRUCT;
   END_VAR
BEGIN
END_DATA_BLOCK

DATA_BLOCK "FG04Actors"   // DB1403
{ S7_Optimized_Access := 'TRUE' }
VERSION : 0.1
   VAR
      AxisZ : "typeActor_2Out2In";
   END_VAR
BEGIN
END_DATA_BLOCK

// folder: 2. Machine/04_FG04/Stepsequences

DATA_BLOCK "InstSq_4.1"   // DB1411
{ S7_Optimized_Access := 'TRUE' }
VERSION : 0.1
// stored: InstanceOfName Sq_4.1
"Sq_4.1"
BEGIN
END_DATA_BLOCK

// folder: 2. Machine/05_FG05

DATA_BLOCK "InstFG05Control"   // DB1500
{ S7_Optimized_Access := 'TRUE' }
VERSION : 0.1
// stored: InstanceOfName FG05Control
"FG05Control"
BEGIN
END_DATA_BLOCK

DATA_BLOCK "FG05Globals"   // DB1502
{ S7_Optimized_Access := 'TRUE' }
VERSION : 0.1
   VAR
      emptying : Bool;   // Zuführung leerfahren / Empty infeed
      SQ1 : Struct
         readyForIndex : Bool;   // Freigabe für den Indexer zum Anheben / Indexer raising enable
         isInHome : Bool;   // Grundstellung vorhanden / Home position reached
      END_STRUCT;
   END_VAR
BEGIN
END_DATA_BLOCK

DATA_BLOCK "FG05Actors"   // DB1503
{ S7_Optimized_Access := 'TRUE' }
VERSION : 0.1
   VAR
      AxisR : "typeActor_2Out2In";
      AxisX : "typeActor_2Out2In";
      AxisZ1 : "typeActor_2Out2In";
      AxisZ2 : "typeActor_2Out2In";
      CapsSourceStopper : "typeActor_2Out1In";
      Gripper : "typeActor_2Out2In";
      Bunker : "typeActor_1Out0In";
      Conveyor : "typeActor_1Out0In";
      Camera : "typeActor_1Out_SimpleCamera";
   END_VAR
BEGIN
END_DATA_BLOCK

// folder: 2. Machine/05_FG05/Stepsequences

DATA_BLOCK "InstSq_5.1"   // DB1511
{ S7_Optimized_Access := 'TRUE' }
VERSION : 0.1
// stored: InstanceOfName Sq_5.1
"Sq_5.1"
BEGIN
END_DATA_BLOCK

// folder: 2. Machine/10_FG_Transport

DATA_BLOCK "InstTransportControl"   // DB2000
{ S7_Optimized_Access := 'TRUE' }
VERSION : 0.1
// stored: InstanceOfName TransportControl
"TransportControl"
BEGIN
END_DATA_BLOCK

DATA_BLOCK "TransportGlobals"   // DB2002
{ S7_Optimized_Access := 'TRUE' }
VERSION : 0.1
   VAR
      Index01 : Struct
         release : Bool;   // Startfreigabe für FG01 von Indexer / Start enable for FG01 from indexer
      END_STRUCT;
      Index02 : Struct
         release : Bool;   // Startfreigabe für FG02 von Indexer / Start enable for FG02 from indexer
      END_STRUCT;
      Index03 : Struct
         release : Bool;   // Startfreigabe für FG03 von Indexer / Start enable for FG03 from indexer
      END_STRUCT;
      Index04 : Struct
         release : Bool;   // Startfreigabe für FG04 von Indexer / Start enable for FG04 from indexer
      END_STRUCT;
      Index05 : Struct
         release : Bool;   // Startfreigabe für FG05 von Indexer / Start enable for FG05 from indexer
      END_STRUCT;
   END_VAR
BEGIN
END_DATA_BLOCK

DATA_BLOCK "TransportActors"   // DB2003
{ S7_Optimized_Access := 'TRUE' }
VERSION : 0.1
   VAR
      Index01_Lift : "typeActor_2Out2In";
      Index01_Stopper : "typeActor_1Out1In";
      Index02_Lift : "typeActor_2Out2In";
      Index02_Stopper : "typeActor_1Out1In";
      Index03_Lift : "typeActor_2Out2In";
      Index03_Stopper : "typeActor_1Out1In";
      Index04_Lift : "typeActor_2Out2In";
      Index04_Stopper : "typeActor_1Out1In";
      Index05_Lift : "typeActor_2Out2In";
      Index05_Stopper : "typeActor_1Out1In";
      Stopper01 : "typeActor_1Out1In";
      Stopper02 : "typeActor_1Out1In";
      Stopper03 : "typeActor_1Out1In";
      Stopper04 : "typeActor_1Out1In";
      Lift01_Lift : "typeActor_2Out2In";
      Lift01_Conv : "typeActor_2Out0In";
      Lift02_Lift : "typeActor_2Out2In";
      Lift02_Conv : "typeActor_2Out0In";
      Transport01_Conv : "typeActor_2Out0In";
      Transport02_Conv : "typeActor_2Out0In";
   END_VAR
BEGIN
END_DATA_BLOCK

// folder: 2. Machine/10_FG_Transport/Stepsequences

DATA_BLOCK "InstSq_Stopper01"   // DB2011
{ S7_Optimized_Access := 'TRUE' }
VERSION : 0.1
// stored: InstanceOfName Sq_Process_Stopper
"Sq_Process_Stopper"
BEGIN
END_DATA_BLOCK

DATA_BLOCK "InstSq_Stopper02"   // DB2012
{ S7_Optimized_Access := 'TRUE' }
VERSION : 0.1
// stored: InstanceOfName Sq_Process_Stopper
"Sq_Process_Stopper"
BEGIN
END_DATA_BLOCK

DATA_BLOCK "InstSq_Stopper03"   // DB2013
{ S7_Optimized_Access := 'TRUE' }
VERSION : 0.1
// stored: InstanceOfName Sq_Process_Stopper
"Sq_Process_Stopper"
BEGIN
END_DATA_BLOCK

DATA_BLOCK "InstSq_Stopper04"   // DB2014
{ S7_Optimized_Access := 'TRUE' }
VERSION : 0.1
// stored: InstanceOfName Sq_Process_Stopper
"Sq_Process_Stopper"
BEGIN
END_DATA_BLOCK

DATA_BLOCK "InstSq_Process_Lift1"   // DB2015
{ S7_Optimized_Access := 'TRUE' }
VERSION : 0.1
// stored: InstanceOfName Sq_Process_Lift
"Sq_Process_Lift"
BEGIN
END_DATA_BLOCK

DATA_BLOCK "InstSq_Process_Lift2"   // DB2016
{ S7_Optimized_Access := 'TRUE' }
VERSION : 0.1
// stored: InstanceOfName Sq_Process_Lift
"Sq_Process_Lift"
BEGIN
END_DATA_BLOCK

DATA_BLOCK "InstSq_Process_Index01"   // DB2017
{ S7_Optimized_Access := 'TRUE' }
VERSION : 0.1
// stored: InstanceOfName Sq_Process_IndexingUnit
"Sq_Process_IndexingUnit"
BEGIN
END_DATA_BLOCK

DATA_BLOCK "InstSq_Process_Index02"   // DB2018
{ S7_Optimized_Access := 'TRUE' }
VERSION : 0.1
// stored: InstanceOfName Sq_Process_IndexingUnit
"Sq_Process_IndexingUnit"
BEGIN
END_DATA_BLOCK

DATA_BLOCK "InstSq_Process_Index03"   // DB2019
{ S7_Optimized_Access := 'TRUE' }
VERSION : 0.1
// stored: InstanceOfName Sq_Process_IndexingUnit
"Sq_Process_IndexingUnit"
BEGIN
END_DATA_BLOCK

DATA_BLOCK "InstSq_Process_Index04"   // DB2020
{ S7_Optimized_Access := 'TRUE' }
VERSION : 0.1
// stored: InstanceOfName Sq_Process_IndexingUnit
"Sq_Process_IndexingUnit"
BEGIN
END_DATA_BLOCK

DATA_BLOCK "InstSq_Process_Index05"   // DB2021
{ S7_Optimized_Access := 'TRUE' }
VERSION : 0.1
// stored: InstanceOfName Sq_Process_IndexingUnit
"Sq_Process_IndexingUnit"
BEGIN
END_DATA_BLOCK

DATA_BLOCK "InstTofRunConveyor1"   // DB2030
{ S7_Optimized_Access := 'TRUE' }
AUTHOR : Simatic
FAMILY : IEC
NAME : IEC_TMR
VERSION : 1.0
// stored: InstanceOfName IEC_TIMER
"IEC_TIMER"
BEGIN
END_DATA_BLOCK

DATA_BLOCK "InstTofRunConveyor2"   // DB2031
{ S7_Optimized_Access := 'TRUE' }
AUTHOR : Simatic
FAMILY : IEC
NAME : IEC_TMR
VERSION : 1.0
// stored: InstanceOfName IEC_TIMER
"IEC_TIMER"
BEGIN
END_DATA_BLOCK

// folder: (top level)

ORGANIZATION_BLOCK "Main"   // OB1, LAD, ProgramCycle
TITLE = "Main Program Sweep (Cycle)" / „Zyklischer Hauptprogrammdurchlauf“
{ S7_Optimized_Access := 'TRUE' }
VERSION : 0.1
   VAR_INPUT
      Initial_Call : Bool;   // Initial call of this OB
      Remanence : Bool;   // =True, if remanent data are available
   END_VAR
BEGIN

REGION Network 1: Inbetriebnahme-Merker / Commissioning flag
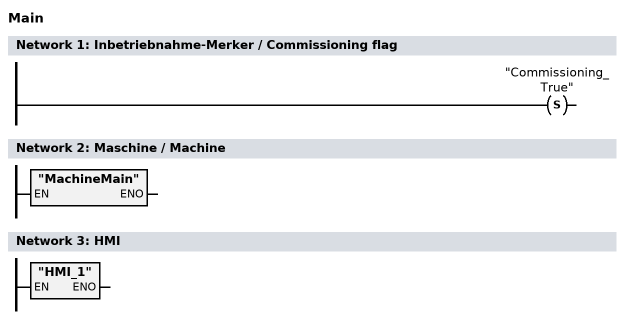
   RUNG wire#powerrail
      S_Coil( "Commissioning_True" )
   END_RUNG
   // the same network as SCL:
   "Commissioning_True" := TRUE;
END_REGION

REGION Network 2: Maschine / Machine
   RUNG wire#powerrail
      "MachineMain"()
   END_RUNG
   // the same network as SCL:
   "MachineMain"();
END_REGION

REGION Network 3: HMI
   RUNG wire#powerrail
      "HMI_1"()
   END_RUNG
   // the same network as SCL:
   "HMI_1"();
END_REGION
END_ORGANIZATION_BLOCK

// folder: 1. HMI/TP700_HMI_1

FUNCTION "HMI_1" : Void   // FC1001, FBD
TITLE = HMI
{ S7_Optimized_Access := 'TRUE' }
VERSION : 0.1
// Ersteller: Andreas Fast Automation
// Kontakt per LinkedIn: https://www.linkedin.com/in/automation-fast-andreas/
// 
// Das Projekt dient zu Demonstrationszwecken und kann frei genutzt werden.
// 
// Bausteinbeschreibung:
// Author: Andreas Fast Automation
// Kontakt per LinkedIn: https://www.linkedin.com/in/automation-fast-andreas/
// 
// This project is intended for demonstration purposes and may be used freely.
// 
// Block description:
BEGIN

REGION Network 1: Steuerung und Anzeige Einrichtbetrieb / Setup mode control and display
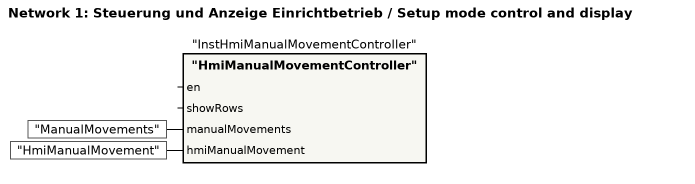
   "InstHmiManualMovementController"(manualMovements := "ManualMovements",   // "HmiManualMovementController"
                           hmiManualMovement := "HmiManualMovement");
END_REGION

REGION Network 2: Anzeige Schrittketteninformationen / Display sequence information
END_REGION
END_FUNCTION

// folder: 2. Machine

FUNCTION "MachineMain" : Void   // FC1000, FBD
TITLE = Maschine / Machine
{ S7_Optimized_Access := 'TRUE' }
VERSION : 0.1
// Ersteller: Andreas Fast Automation
// Kontakt per LinkedIn: https://www.linkedin.com/in/automation-fast-andreas/
// 
// Das Projekt dient zu Demonstrationszwecken und kann frei genutzt werden.
// Author: Andreas Fast Automation
// Kontakt per LinkedIn: https://www.linkedin.com/in/automation-fast-andreas/
// 
// This project is intended for demonstration purposes and may be used freely.
BEGIN

REGION Network 1: Maschine / Machine
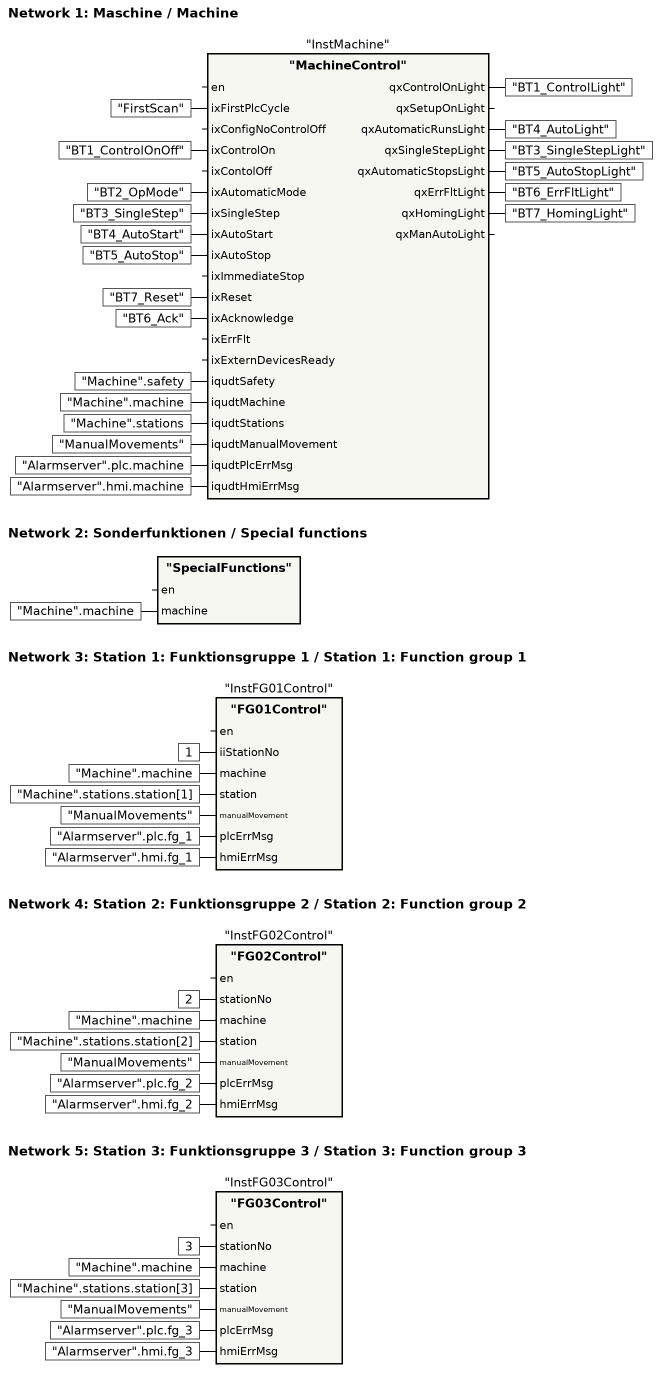
   "InstMachine"(ixFirstPlcCycle := "FirstScan",   // "MachineControl"
                 ixControlOn := "BT1_ControlOnOff",
                 ixAutomaticMode := "BT2_OpMode",
                 ixSingleStep := "BT3_SingleStep",
                 ixAutoStart := "BT4_AutoStart",
                 ixAutoStop := "BT5_AutoStop",
                 ixReset := "BT7_Reset",
                 ixAcknowledge := "BT6_Ack",
                 iqudtSafety := "Machine".safety,
                 iqudtMachine := "Machine".machine,
                 iqudtStations := "Machine".stations,
                 iqudtManualMovement := "ManualMovements",
                 iqudtPlcErrMsg := "Alarmserver".plc.machine,
                 iqudtHmiErrMsg := "Alarmserver".hmi.machine,
                 qxControlOnLight => "BT1_ControlLight",
                 qxAutomaticRunsLight => "BT4_AutoLight",
                 qxSingleStepLight => "BT3_SingleStepLight",
                 qxAutomaticStopsLight => "BT5_AutoStopLight",
                 qxErrFltLight => "BT6_ErrFltLight",
                 qxHomingLight => "BT7_HomingLight");
END_REGION

REGION Network 2: Sonderfunktionen / Special functions
   "SpecialFunctions"(machine := "Machine".machine);
END_REGION

REGION Network 3: Station 1: Funktionsgruppe 1 / Station 1: Function group 1
   "InstFG01Control"(iiStationNo := 1,   // "FG01Control"
                     machine := "Machine".machine,
                     station := "Machine".stations.station[1],
                     manualMovement := "ManualMovements",
                     plcErrMsg := "Alarmserver".plc.fg_1,
                     hmiErrMsg := "Alarmserver".hmi.fg_1);
END_REGION

REGION Network 4: Station 2: Funktionsgruppe 2 / Station 2: Function group 2
   "InstFG02Control"(stationNo := 2,   // "FG02Control"
                     machine := "Machine".machine,
                     station := "Machine".stations.station[2],
                     manualMovement := "ManualMovements",
                     plcErrMsg := "Alarmserver".plc.fg_2,
                     hmiErrMsg := "Alarmserver".hmi.fg_2);
END_REGION

REGION Network 5: Station 3: Funktionsgruppe 3 / Station 3: Function group 3
   "InstFG03Control"(stationNo := 3,   // "FG03Control"
                     machine := "Machine".machine,
                     station := "Machine".stations.station[3],
                     manualMovement := "ManualMovements",
                     plcErrMsg := "Alarmserver".plc.fg_3,
                     hmiErrMsg := "Alarmserver".hmi.fg_3);
END_REGION

REGION Network 6: Station 4: Funktionsgruppe 4 / Station 4: Function group 4
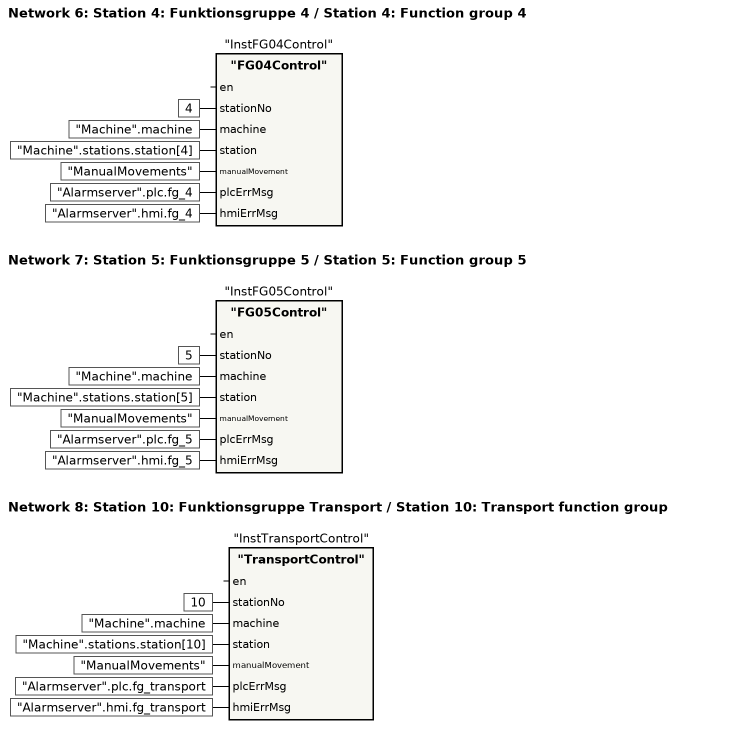
   "InstFG04Control"(stationNo := 4,   // "FG04Control"
                     machine := "Machine".machine,
                     station := "Machine".stations.station[4],
                     manualMovement := "ManualMovements",
                     plcErrMsg := "Alarmserver".plc.fg_4,
                     hmiErrMsg := "Alarmserver".hmi.fg_4);
END_REGION

REGION Network 7: Station 5: Funktionsgruppe 5 / Station 5: Function group 5
   "InstFG05Control"(stationNo := 5,   // "FG05Control"
                     machine := "Machine".machine,
                     station := "Machine".stations.station[5],
                     manualMovement := "ManualMovements",
                     plcErrMsg := "Alarmserver".plc.fg_5,
                     hmiErrMsg := "Alarmserver".hmi.fg_5);
END_REGION

REGION Network 8: Station 10: Funktionsgruppe Transport / Station 10: Transport function group
   "InstTransportControl"(stationNo := 10,   // "TransportControl"
                          machine := "Machine".machine,
                          station := "Machine".stations.station[10],
                          manualMovement := "ManualMovements",
                          plcErrMsg := "Alarmserver".plc.fg_transport,
                          hmiErrMsg := "Alarmserver".hmi.fg_transport);
END_REGION
END_FUNCTION

FUNCTION "SpecialFunctions" : Void   // FC1090, LAD
TITLE = Sonderfunktionen / Special functions
{ S7_Optimized_Access := 'TRUE' }
VERSION : 0.1
   VAR_IN_OUT
      machine : "typeMachine";
   END_VAR
BEGIN

REGION Network 1: Ampel / Signal tower
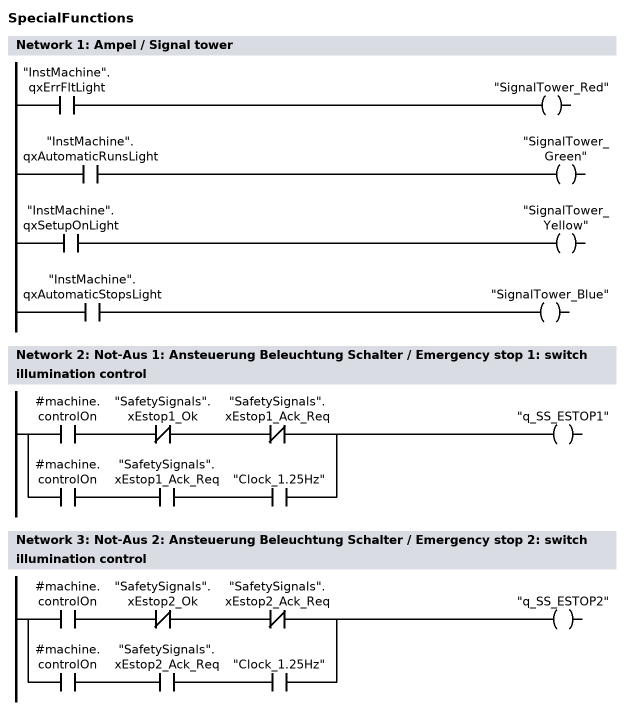
   RUNG wire#powerrail
      Contact( "InstMachine".qxErrFltLight )
      Coil( "SignalTower_Red" )
   END_RUNG
   RUNG wire#powerrail
      Contact( "InstMachine".qxAutomaticRunsLight )
      Coil( "SignalTower_Green" )
   END_RUNG
   RUNG wire#powerrail
      Contact( "InstMachine".qxSetupOnLight )
      Coil( "SignalTower_Yellow" )
   END_RUNG
   RUNG wire#powerrail
      Contact( "InstMachine".qxAutomaticStopsLight )
      Coil( "SignalTower_Blue" )
   END_RUNG
   // the same network as SCL:
   "SignalTower_Red" := "InstMachine".qxErrFltLight;
   "SignalTower_Green" := "InstMachine".qxAutomaticRunsLight;
   "SignalTower_Yellow" := "InstMachine".qxSetupOnLight;
   "SignalTower_Blue" := "InstMachine".qxAutomaticStopsLight;
END_REGION

REGION Network 2: Not-Aus 1: Ansteuerung Beleuchtung Schalter / Emergency stop 1: switch illumination control
   RUNG wire#powerrail
      Contact( #machine.controlOn )
      I_Contact( "SafetySignals".xEstop1_Ok )
      I_Contact( "SafetySignals".xEstop1_Ack_Req )
      wire#w1
      Coil( "q_SS_ESTOP1" )
   END_RUNG
   RUNG wire#powerrail
      Contact( #machine.controlOn )
      Contact( "SafetySignals".xEstop1_Ack_Req )
      Contact( "Clock_1.25Hz" )
   END_RUNG wire#w1
   // the same network as SCL:
   "q_SS_ESTOP1" := (#machine.controlOn AND NOT "SafetySignals".xEstop1_Ok AND NOT "SafetySignals".xEstop1_Ack_Req) OR (#machine.controlOn AND "SafetySignals".xEstop1_Ack_Req AND "Clock_1.25Hz");
END_REGION

REGION Network 3: Not-Aus 2: Ansteuerung Beleuchtung Schalter / Emergency stop 2: switch illumination control
   RUNG wire#powerrail
      Contact( #machine.controlOn )
      I_Contact( "SafetySignals".xEstop2_Ok )
      I_Contact( "SafetySignals".xEstop2_Ack_Req )
      wire#w1
      Coil( "q_SS_ESTOP2" )
   END_RUNG
   RUNG wire#powerrail
      Contact( #machine.controlOn )
      Contact( "SafetySignals".xEstop2_Ack_Req )
      Contact( "Clock_1.25Hz" )
   END_RUNG wire#w1
   // the same network as SCL:
   "q_SS_ESTOP2" := (#machine.controlOn AND NOT "SafetySignals".xEstop2_Ok AND NOT "SafetySignals".xEstop2_Ack_Req) OR (#machine.controlOn AND "SafetySignals".xEstop2_Ack_Req AND "Clock_1.25Hz");
END_REGION
END_FUNCTION

// folder: 2. Machine/00_Alarms and Messages

FUNCTION "MachineAlarms" : Void   // FC1009, LAD
TITLE = Störmeldungen Maschine / Machine fault messages
{ S7_Optimized_Access := 'TRUE' }
VERSION : 0.1
// Ersteller: Andreas Fast Automation
// Kontakt per LinkedIn: https://www.linkedin.com/in/automation-fast-andreas/
// 
// Das Projekt dient zu Demonstrationszwecken und kann frei genutzt werden.
// 
// Bausteinbeschreibung: 
// Störmeldungen werden über die Quittierung zurückgesetzt.
// Author: Andreas Fast Automation
// Kontakt per LinkedIn: https://www.linkedin.com/in/automation-fast-andreas/
// 
// This project is intended for demonstration purposes and may be used freely.
// 
// Block description:
// Fault messages are reset by acknowledgement.
   VAR_IN_OUT
      machine : "typeMachine";
      alarms : "typePlcErrors";
   END_VAR
BEGIN

REGION Network 1: Initialisierung für die Einrichtbewegungen ist fehlerhaft / Setup movement initialisation failed
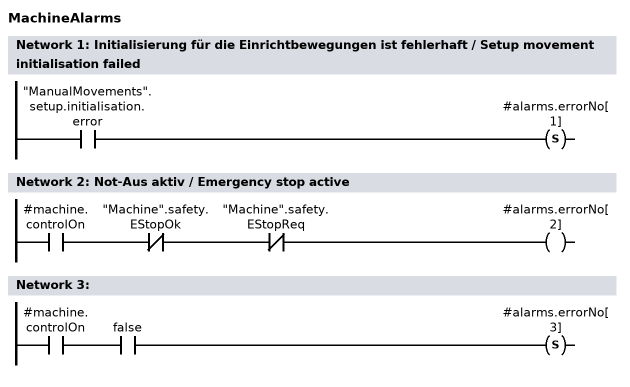
   RUNG wire#powerrail
      Contact( "ManualMovements".setup.initialisation.error )
      S_Coil( #alarms.errorNo[1] )
   END_RUNG
   // the same network as SCL:
   IF "ManualMovements".setup.initialisation.error THEN #alarms.errorNo[1] := TRUE; END_IF;
END_REGION

REGION Network 2: Not-Aus aktiv / Emergency stop active
   RUNG wire#powerrail
      Contact( #machine.controlOn )
      I_Contact( "Machine".safety.EStopOk )
      I_Contact( "Machine".safety.EStopReq )
      Coil( #alarms.errorNo[2] )
   END_RUNG
   // the same network as SCL:
   #alarms.errorNo[2] := #machine.controlOn AND NOT "Machine".safety.EStopOk AND NOT "Machine".safety.EStopReq;
END_REGION

REGION Network 3
   RUNG wire#powerrail
      Contact( #machine.controlOn )
      Contact( false )
      S_Coil( #alarms.errorNo[3] )
   END_RUNG
   // the same network as SCL:
   IF #machine.controlOn AND false THEN #alarms.errorNo[3] := TRUE; END_IF;
END_REGION
END_FUNCTION

FUNCTION "MachineMessages" : Void   // FC1010, LAD
TITLE = Meldungen Maschine / Machine messages
{ S7_Optimized_Access := 'TRUE' }
VERSION : 0.1
// Ersteller: Andreas Fast Automation
// Kontakt per LinkedIn: https://www.linkedin.com/in/automation-fast-andreas/
// 
// Das Projekt dient zu Demonstrationszwecken und kann frei genutzt werden.
// 
// Bausteinbeschreibung: 
// Störmeldungen werden über die Quittierung zurückgesetzt.
// Author: Andreas Fast Automation
// Kontakt per LinkedIn: https://www.linkedin.com/in/automation-fast-andreas/
// 
// This project is intended for demonstration purposes and may be used freely.
// 
// Block description:
// Fault messages are reset by acknowledgement.
   VAR_IN_OUT
      machine : "typeMachine";
      messages : "typePlcMessages";
   END_VAR
BEGIN

REGION Network 1: Maschine ist ausgeschaltet / Machine switched off
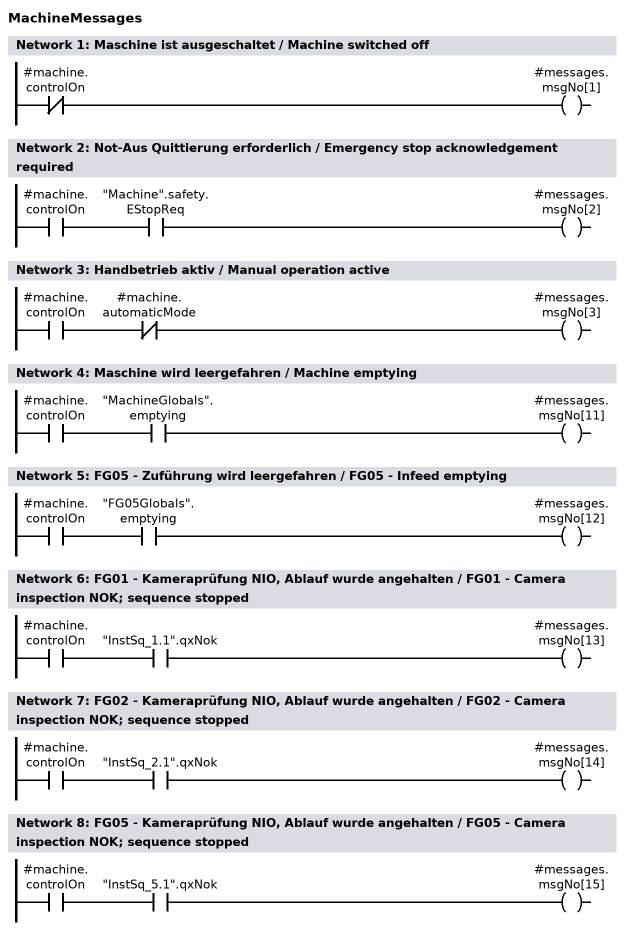
   RUNG wire#powerrail
      I_Contact( #machine.controlOn )
      Coil( #messages.msgNo[1] )
   END_RUNG
   // the same network as SCL:
   #messages.msgNo[1] := NOT #machine.controlOn;
END_REGION

REGION Network 2: Not-Aus Quittierung erforderlich / Emergency stop acknowledgement required
   RUNG wire#powerrail
      Contact( #machine.controlOn )
      Contact( "Machine".safety.EStopReq )
      Coil( #messages.msgNo[2] )
   END_RUNG
   // the same network as SCL:
   #messages.msgNo[2] := #machine.controlOn AND "Machine".safety.EStopReq;
END_REGION

REGION Network 3: Handbetrieb aktiv / Manual operation active
   RUNG wire#powerrail
      Contact( #machine.controlOn )
      I_Contact( #machine.automaticMode )
      Coil( #messages.msgNo[3] )
   END_RUNG
   // the same network as SCL:
   #messages.msgNo[3] := #machine.controlOn AND NOT #machine.automaticMode;
END_REGION

REGION Network 4: Maschine wird leergefahren / Machine emptying
   RUNG wire#powerrail
      Contact( #machine.controlOn )
      Contact( "MachineGlobals".emptying )
      Coil( #messages.msgNo[11] )
   END_RUNG
   // the same network as SCL:
   #messages.msgNo[11] := #machine.controlOn AND "MachineGlobals".emptying;
END_REGION

REGION Network 5: FG05 - Zuführung wird leergefahren / FG05 - Infeed emptying
   RUNG wire#powerrail
      Contact( #machine.controlOn )
      Contact( "FG05Globals".emptying )
      Coil( #messages.msgNo[12] )
   END_RUNG
   // the same network as SCL:
   #messages.msgNo[12] := #machine.controlOn AND "FG05Globals".emptying;
END_REGION

REGION Network 6: FG01 - Kameraprüfung NIO, Ablauf wurde angehalten / FG01 - Camera inspection NOK; sequence stopped
   RUNG wire#powerrail
      Contact( #machine.controlOn )
      Contact( "InstSq_1.1".qxNok )
      Coil( #messages.msgNo[13] )
   END_RUNG
   // the same network as SCL:
   #messages.msgNo[13] := #machine.controlOn AND "InstSq_1.1".qxNok;
END_REGION

REGION Network 7: FG02 - Kameraprüfung NIO, Ablauf wurde angehalten / FG02 - Camera inspection NOK; sequence stopped
   RUNG wire#powerrail
      Contact( #machine.controlOn )
      Contact( "InstSq_2.1".qxNok )
      Coil( #messages.msgNo[14] )
   END_RUNG
   // the same network as SCL:
   #messages.msgNo[14] := #machine.controlOn AND "InstSq_2.1".qxNok;
END_REGION

REGION Network 8: FG05 - Kameraprüfung NIO, Ablauf wurde angehalten / FG05 - Camera inspection NOK; sequence stopped
   RUNG wire#powerrail
      Contact( #machine.controlOn )
      Contact( "InstSq_5.1".qxNok )
      Coil( #messages.msgNo[15] )
   END_RUNG
   // the same network as SCL:
   #messages.msgNo[15] := #machine.controlOn AND "InstSq_5.1".qxNok;
END_REGION
END_FUNCTION

// folder: 2. Machine/01_FG01

FUNCTION_BLOCK "FG01Control"   // FB1100, FBD
TITLE = Station 1 Hauptaufruf / Station 1 main call
{ S7_Optimized_Access := 'TRUE' }
VERSION : 0.1
// Ersteller: Andreas Fast Automation
// Kontakt per LinkedIn: https://www.linkedin.com/in/automation-fast-andreas/
// 
// Das Projekt dient zu Demonstrationszwecken und kann frei genutzt werden.
// 
// Bausteinbeschreibung:
// Author: Andreas Fast Automation
// Kontakt per LinkedIn: https://www.linkedin.com/in/automation-fast-andreas/
// 
// This project is intended for demonstration purposes and may be used freely.
// 
// Block description:
   VAR_INPUT
      iiStationNo : Int := 1;   // Stationsnummer / Station number
   END_VAR
   VAR_IN_OUT
      machine : "typeMachine";
      station : "typeStation";
      manualMovement : "typeManualMovements";
      plcErrMsg : "typePlcErrMsg";
      hmiErrMsg : "typeHmiErrMsg";
   END_VAR
   VAR
      instStationControl : "StationControl";
      instActorControl : "FG01ActorControl";
      instStationState : "StationState";
      sinstStationCycleTime : "StationCycleTime";
   END_VAR
   VAR_TEMP
      tempSafetyOk : Bool;
   END_VAR
BEGIN

REGION Network 1: Stationssteuerung / Station control
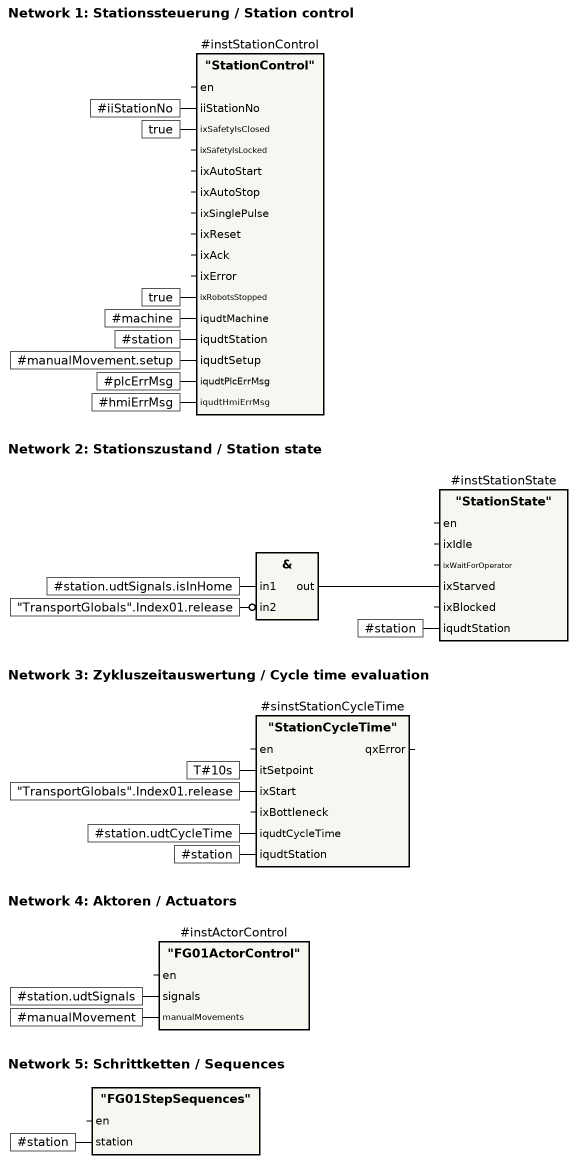
   #instStationControl(iiStationNo := #iiStationNo,   // "StationControl"
                       ixSafetyIsClosed := true,
                       ixRobotsStopped := true,
                       iqudtMachine := #machine,
                       iqudtStation := #station,
                       iqudtSetup := #manualMovement.setup,
                       iqudtPlcErrMsg := #plcErrMsg,
                       iqudtHmiErrMsg := #hmiErrMsg);
END_REGION

REGION Network 2: Stationszustand / Station state
   #instStationState(ixStarved := #station.udtSignals.isInHome AND NOT "TransportGlobals".Index01.release,   // "StationState"
                     iqudtStation := #station);
END_REGION

REGION Network 3: Zykluszeitauswertung / Cycle time evaluation
   #sinstStationCycleTime(itSetpoint := T#10s,   // "StationCycleTime"
                          ixStart := "TransportGlobals".Index01.release,
                          iqudtCycleTime := #station.udtCycleTime,
                          iqudtStation := #station);
END_REGION

REGION Network 4: Aktoren / Actuators
   #instActorControl(signals := #station.udtSignals, manualMovements := #manualMovement);   // "FG01ActorControl"
END_REGION

REGION Network 5: Schrittketten / Sequences
   "FG01StepSequences"(station := #station);
END_REGION
END_FUNCTION_BLOCK

FUNCTION_BLOCK "FG01ActorControl"   // FB1102, FBD
TITLE = Aktoransteuerung / Actuator control
{ S7_Optimized_Access := 'TRUE' }
VERSION : 0.1
// Ersteller: Andreas Fast Automation
// Kontakt per LinkedIn: https://www.linkedin.com/in/automation-fast-andreas/
// 
// Das Projekt dient zu Demonstrationszwecken und kann frei genutzt werden.
// 
// Bausteinbeschreibung:
// Author: Andreas Fast Automation
// Kontakt per LinkedIn: https://www.linkedin.com/in/automation-fast-andreas/
// 
// This project is intended for demonstration purposes and may be used freely.
// 
// Block description:
   VAR_IN_OUT
      signals : "typeStationSignals";
      manualMovements : "typeManualMovements";
   END_VAR
   VAR
      sinstGripper : "Cylinder_2Out2In";
      sinstPlattform : "Cylinder_2Out2In";
      sinstReaderWindow : "Cylinder_2Out1In";
      sinstLasermark : "Cylinder_1Out0In";
      sinstGate_1 : "Cylinder_1Out2In";
      sinstGate_2 : "Cylinder_1Out2In";
      sinstCamera : "Actor_1Out_SimpleCamera";
   END_VAR
BEGIN

REGION Network 1: Greifer / Gripper
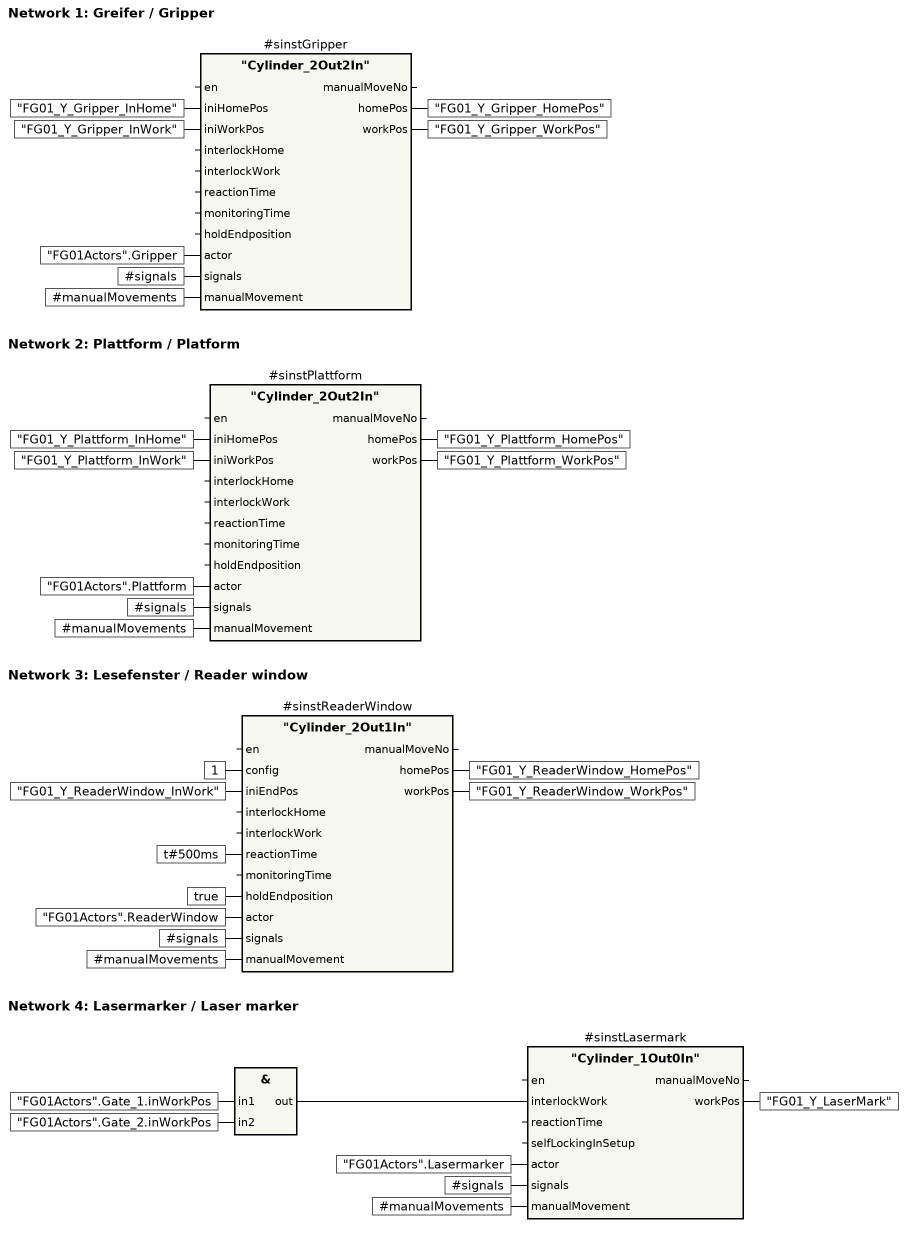
   #sinstGripper(iniHomePos := "FG01_Y_Gripper_InHome",   // "Cylinder_2Out2In"
                 iniWorkPos := "FG01_Y_Gripper_InWork",
                 actor := "FG01Actors".Gripper,
                 signals := #signals,
                 manualMovement := #manualMovements,
                 homePos => "FG01_Y_Gripper_HomePos",
                 workPos => "FG01_Y_Gripper_WorkPos");
END_REGION

REGION Network 2: Plattform / Platform
   #sinstPlattform(iniHomePos := "FG01_Y_Plattform_InHome",   // "Cylinder_2Out2In"
                   iniWorkPos := "FG01_Y_Plattform_InWork",
                   actor := "FG01Actors".Plattform,
                   signals := #signals,
                   manualMovement := #manualMovements,
                   homePos => "FG01_Y_Plattform_HomePos",
                   workPos => "FG01_Y_Plattform_WorkPos");
END_REGION

REGION Network 3: Lesefenster / Reader window
   #sinstReaderWindow(config := 1,   // "Cylinder_2Out1In"
                      iniEndPos := "FG01_Y_ReaderWindow_InWork",
                      reactionTime := t#500ms,
                      holdEndposition := true,
                      actor := "FG01Actors".ReaderWindow,
                      signals := #signals,
                      manualMovement := #manualMovements,
                      homePos => "FG01_Y_ReaderWindow_HomePos",
                      workPos => "FG01_Y_ReaderWindow_WorkPos");
END_REGION

REGION Network 4: Lasermarker / Laser marker
   #sinstLasermark(interlockWork := "FG01Actors".Gate_1.inWorkPos AND "FG01Actors".Gate_2.inWorkPos,   // "Cylinder_1Out0In"
                   actor := "FG01Actors".Lasermarker,
                   signals := #signals,
                   manualMovement := #manualMovements,
                   workPos => "FG01_Y_LaserMark");
END_REGION

REGION Network 5: Tor 1 / Gate 1
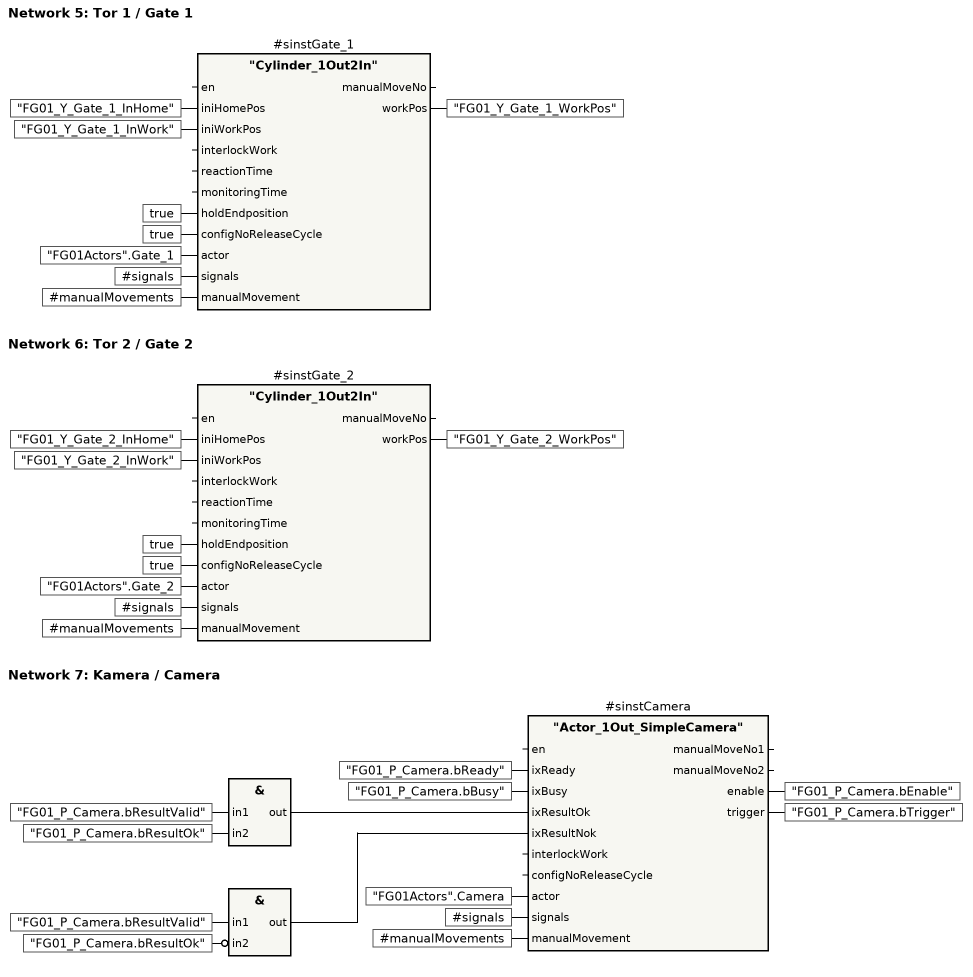
   #sinstGate_1(iniHomePos := "FG01_Y_Gate_1_InHome",   // "Cylinder_1Out2In"
                iniWorkPos := "FG01_Y_Gate_1_InWork",
                holdEndposition := true,
                configNoReleaseCycle := true,
                actor := "FG01Actors".Gate_1,
                signals := #signals,
                manualMovement := #manualMovements,
                workPos => "FG01_Y_Gate_1_WorkPos");
END_REGION

REGION Network 6: Tor 2 / Gate 2
   #sinstGate_2(iniHomePos := "FG01_Y_Gate_2_InHome",   // "Cylinder_1Out2In"
                iniWorkPos := "FG01_Y_Gate_2_InWork",
                holdEndposition := true,
                configNoReleaseCycle := true,
                actor := "FG01Actors".Gate_2,
                signals := #signals,
                manualMovement := #manualMovements,
                workPos => "FG01_Y_Gate_2_WorkPos");
END_REGION

REGION Network 7: Kamera / Camera
   #sinstCamera(ixReady := "FG01_P_Camera.bReady",   // "Actor_1Out_SimpleCamera"
                ixBusy := "FG01_P_Camera.bBusy",
                ixResultOk := "FG01_P_Camera.bResultValid" AND "FG01_P_Camera.bResultOk",
                ixResultNok := "FG01_P_Camera.bResultValid" AND NOT "FG01_P_Camera.bResultOk",
                actor := "FG01Actors".Camera,
                signals := #signals,
                manualMovement := #manualMovements,
                enable => "FG01_P_Camera.bEnable",
                trigger => "FG01_P_Camera.bTrigger");
END_REGION
END_FUNCTION_BLOCK

// folder: 2. Machine/01_FG01/Stepsequences

FUNCTION_BLOCK "Sq_1.1"   // FB1111, GRAPH_PLUS
{ S7_Optimized_Access := 'TRUE' }
VERSION : 0.1
   VAR_INPUT
      OFF_SQ : Bool := false;   // Kette ausschalten
      INIT_SQ : Bool := false;   // Kette in Initialzustand versetzen
      ACK_EF : Bool := false;   // Alle Fehler und Störungen quittieren
      S_PREV : Bool := false;   // Vorherigen Schritt am Parameter S_NO ausgeben
      S_NEXT : Bool := false;   // Nächsten Schritt am Parameter S_NO anzeigen
      SW_AUTO : Bool := false;   // Automatischer Betrieb
      SW_TAP : Bool := false;   // Halbautomatisch/Weiterschalten mit Transition
      SW_TOP : Bool := false;   // Halbautomatisch/Ignoriere Transition
      SW_MAN : Bool := false;   // Handbetrieb
      S_SEL : Int := 0;   // Schritt auswählen, der an S_NO ausgegeben werden soll
      S_ON : Bool := false;   // Schritt aktivieren, der an Parameter S_NO anliegt
      S_OFF : Bool := false;   // Schritt deaktivieren, der an Parameter S_NO anliegt
      T_PUSH : Bool := false;   // Schaltfreigabe für Transition im halbautomatischen Betrieb
      itMaxRuntime : Time := t#10s;   // Maximale Laufzeit für diesen Prozess / Maximum execution time for this process
   END_VAR
   VAR_OUTPUT
      S_NO : Int := 0;   // Schrittnummer
      S_MORE : Bool := false;   // Weitere Schritte sind vorhanden und können in S_NO angezeigt werden.
      S_ACTIVE : Bool := false;   // Schritt, der an Parameter S_NO angezeigt wird, ist aktiv
      ERR_FLT : Bool := false;   // Sammelfehler Interlock oder Supervision
      AUTO_ON : Bool := false;   // Automatischer Betrieb eingeschaltet
      TAP_ON : Bool := false;   // Halbautomatischer Betrieb/Schritt mit Transition eingeschaltet
      TOP_ON : Bool := false;   // Halbautomatischer Betrieb/Ignoriere Transition eingeschaltet
      MAN_ON : Bool := false;   // Handbetrieb eingeschaltet
      qxIsActive : Bool;   // Schrittkette läuft / Sequence running
      qxIsInHome : Bool;   // steht in Grundstellung / in home position
      qxNok : Bool;   // NIO Teil / NOK part
   END_VAR
   VAR_IN_OUT
      signals : "typeStationSignals";   // Stationssteuersignale / Station control signals
      sq : "typeStepSequence";   // Schrittkettensteuersignale / Sequence control signals
   END_VAR
   VAR
      sstReleaseCycle : Struct
         ErrorAck : Bool;
         No_LastCycle : Int;
         T : Time;   // Aktive Zeit des ReleaseCycle / Active time of ReleaseCycle
         Tck : Time;
         TckPrev : Time;
      END_STRUCT;
      HMI_INFO : Array[0..8] of UInt;
      IF_PAR : G7_IfParPlus_V6;
      RT_DATA : G7_RTDataPlus_V6;   // Interner Datenbereich
      Automatikablauf : G7_TransitionPlus_V6;   // Transitionsstruktur
      Freigabe : G7_TransitionPlus_V6;   // Transitionsstruktur
      Trans3 : G7_TransitionPlus_V6;   // Transitionsstruktur
      Fertig : G7_TransitionPlus_V6;   // Transitionsstruktur
      Grundstellungsfahrt : G7_TransitionPlus_V6;   // Transitionsstruktur
      GST_Aktiv : G7_TransitionPlus_V6;   // Transitionsstruktur
      GST_Beendet : G7_TransitionPlus_V6;   // Transitionsstruktur
      Beendet : G7_TransitionPlus_V6;   // Transitionsstruktur
      DoneToIndexer : G7_TransitionPlus_V6;   // Transitionsstruktur / Transition structure
      TriggerIsSet : G7_TransitionPlus_V6;   // Transition structure / Transitionsstruktur
      CamIsDone : G7_TransitionPlus_V6;   // Transition structure / Transitionsstruktur
      TriggerIsReseted : G7_TransitionPlus_V6;   // Transition structure / Transitionsstruktur
      GS_GripperInHome : G7_TransitionPlus_V6;   // Transitionsstruktur / Transition structure
      GS_PlattformInHome : G7_TransitionPlus_V6;   // Transitionsstruktur / Transition structure
      GS_ReaderWindowInHome : G7_TransitionPlus_V6;   // Transitionsstruktur / Transition structure
      PlattformIsInWork : G7_TransitionPlus_V6;   // Transitionsstruktur / Transition structure
      ReaderWindowInWork : G7_TransitionPlus_V6;   // Transition structure / Transitionsstruktur
      GripperInWork : G7_TransitionPlus_V6;   // Transitionsstruktur / Transition structure
      GripperInHome : G7_TransitionPlus_V6;   // Transitionsstruktur / Transition structure
      PlattformIsInWork_1 : G7_TransitionPlus_V6;   // Transitionsstruktur / Transition structure
      ReaderWindowInHome : G7_TransitionPlus_V6;   // Transitionsstruktur / Transition structure
      JogT3 : G7_TransitionPlus_V6;   // Transitionsstruktur / Transition structure
      JogT4 : G7_TransitionPlus_V6;   // Transitionsstruktur / Transition structure
      JogT1 : G7_TransitionPlus_V6;   // Transition structure / Transitionsstruktur
      JogT7 : G7_TransitionPlus_V6;   // Transitionsstruktur / Transition structure
      LaserDone : G7_TransitionPlus_V6;   // Transitionsstruktur / Transition structure
      JogT8 : G7_TransitionPlus_V6;   // Transitionsstruktur / Transition structure
      GatesClosed : G7_TransitionPlus_V6;   // Transition structure / Transitionsstruktur
      JogT5 : G7_TransitionPlus_V6;   // Transition structure / Transitionsstruktur
      JogT9 : G7_TransitionPlus_V6;   // Transition structure / Transitionsstruktur
      GatesOpened : G7_TransitionPlus_V6;   // Transition structure / Transitionsstruktur
      JogT6 : G7_TransitionPlus_V6;   // Transition structure / Transitionsstruktur
      GS_GatesOpened : G7_TransitionPlus_V6;   // Transition structure / Transitionsstruktur
      LaserIsOn : G7_TransitionPlus_V6;   // Transition structure / Transitionsstruktur
      LaserIsOff : G7_TransitionPlus_V6;   // Transition structure / Transitionsstruktur
      JogT2 : G7_TransitionPlus_V6;   // Transition structure / Transitionsstruktur
      "Result Ok" : G7_TransitionPlus_V6;   // Transition structure / Transitionsstruktur
      "Result Nok" : G7_TransitionPlus_V6;   // Transition structure / Transitionsstruktur
      NIO_Quittiert : G7_TransitionPlus_V6;   // Transition structure / Transitionsstruktur
      Initialschritt : G7_StepPlus_V6;   // Schrittstruktur
      Grundstellung : G7_StepPlus_V6;   // Schrittstruktur
      SK_läuft : G7_StepPlus_V6;   // Schrittstruktur
      Fertigmeldung : G7_StepPlus_V6;   // Schrittstruktur
      "Start Grundstellungsfahrt" : G7_StepPlus_V6;   // Schrittstruktur
      "Fertig Grundstellungsfahrt" : G7_StepPlus_V6;   // Schrittstruktur
      Ende : G7_StepPlus_V6;   // Schrittstruktur
      ResetRelease : G7_StepPlus_V6;   // Schrittstruktur / Step structure
      Set_Trigger : G7_StepPlus_V6;   // Step structure / Schrittstruktur
      Wait_Busy_Done : G7_StepPlus_V6;   // Step structure / Schrittstruktur
      Reset_Trigger : G7_StepPlus_V6;   // Step structure / Schrittstruktur
      GS_GripperHome : G7_StepPlus_V6;   // Schrittstruktur / Step structure
      GS_PlattformHome : G7_StepPlus_V6;   // Schrittstruktur / Step structure
      GS_ReaderWindowHome : G7_StepPlus_V6;   // Schrittstruktur / Step structure
      PlattformToWork : G7_StepPlus_V6;   // Schrittstruktur / Step structure
      ReaderWindowToWork : G7_StepPlus_V6;   // Step structure / Schrittstruktur
      GripperToWork : G7_StepPlus_V6;   // Schrittstruktur / Step structure
      GripperToHome : G7_StepPlus_V6;   // Schrittstruktur / Step structure
      PlattformToHome : G7_StepPlus_V6;   // Schrittstruktur / Step structure
      ReaderWindowToHome : G7_StepPlus_V6;   // Schrittstruktur / Step structure
      JogS3 : G7_StepPlus_V6;   // Schrittstruktur / Step structure
      JogS4 : G7_StepPlus_V6;   // Schrittstruktur / Step structure
      JogS1 : G7_StepPlus_V6;   // Step structure / Schrittstruktur
      JogS7 : G7_StepPlus_V6;   // Schrittstruktur / Step structure
      Laser : G7_StepPlus_V6;   // Schrittstruktur / Step structure
      JogS8 : G7_StepPlus_V6;   // Schrittstruktur / Step structure
      CloseGates : G7_StepPlus_V6;   // Step structure / Schrittstruktur
      JogS5 : G7_StepPlus_V6;   // Step structure / Schrittstruktur
      JogS9 : G7_StepPlus_V6;   // Step structure / Schrittstruktur
      OpenGates : G7_StepPlus_V6;   // Step structure / Schrittstruktur
      JogS6 : G7_StepPlus_V6;   // Step structure / Schrittstruktur
      GS_OpenGates : G7_StepPlus_V6;   // Step structure / Schrittstruktur
      CheckLaserOn : G7_StepPlus_V6;   // Step structure / Schrittstruktur
      JogS2 : G7_StepPlus_V6;   // Step structure / Schrittstruktur
      Check_Result : G7_StepPlus_V6;   // Step structure / Schrittstruktur
      NIO : G7_StepPlus_V6;   // Step structure / Schrittstruktur
      SINI : Array[0..1] of USInt;
      LSTT : Array[0..38] of USInt;
      ATAJ : Array[0..38] of USInt;
      ATAB : Array[0..38] of USInt;
      PSTT : Array[0..38] of USInt;
      NSTT : Array[0..38] of USInt;
      ASSJ : Array[0..35] of USInt;
      ASSB : Array[0..35] of USInt;
      PTTS : Array[0..35] of USInt;
      NTTS : Array[0..35] of USInt;
      SW_SQTS : Array[0..35] of USInt;
      SWITCH : Array[0..7] of USInt;
      TVX : Array[0..7] of USInt;
      TTX : Array[0..7] of USInt;
      TSX : Array[0..1] of USInt;
      S00X : Array[0..1] of USInt;
      SOFFX : Array[0..1] of USInt;
      SONX : Array[0..1] of USInt;
      SAX : Array[0..1] of USInt;
      SERRX : Array[0..36] of USInt;
      SMX : Array[0..36] of USInt;
      S0X : Array[0..36] of USInt;
      S1X : Array[0..36] of USInt;
      IL_ALARM_INST : Diag_Alarm;
      SUP_ALARM_INST : Diag_Alarm;
      STEP_TIME_ALARM_INST : Diag_Alarm;
      IEC_TIMER_INST : IEC_TIMER;
      TRANSACTION_FLAG : Bool := false;
   END_VAR
   VAR_TEMP
      txStartCondition : Bool;
      tdTckDiff : DInt;
   END_VAR
   VAR_TEMP   // added for the SCL form of the ladder/FBD networks
      _w1 : Bool;
      _w2 : Bool;
   END_VAR
   // SINI[0] := 2;
   // LSTT[0] := 255;
   // LSTT[1] := 255;
   // LSTT[2] := 255;
   // LSTT[3] := 255;
   // LSTT[4] := 255;
   // LSTT[5] := 255;
   // LSTT[6] := 255;
   // LSTT[7] := 1;
   // ATAJ[1] := 1;
   // ATAJ[2] := 2;
   // ATAJ[3] := 6;
   // ATAJ[4] := 4;
   // ATAJ[5] := 5;
   // ATAJ[6] := 3;
   // ATAJ[7] := 7;
   // ATAB[0] := 4;
   // ATAB[1] := 1;
   // ATAB[2] := 2;
   // ATAB[3] := 3;
   // ATAB[5] := 5;
   // ATAB[6] := 6;
   // ATAB[7] := 7;
   // PSTT[1] := 1;
   // PSTT[2] := 2;
   // PSTT[3] := 3;
   // PSTT[5] := 4;
   // PSTT[6] := 5;
   // PSTT[7] := 6;
   // NSTT[0] := 1;
   // NSTT[1] := 2;
   // NSTT[2] := 15;
   // NSTT[3] := 6;
   // NSTT[4] := 4;
   // NSTT[5] := 11;
   // NSTT[6] := 6;
   // NSTT[7] := 1;
   // ASSJ[1] := 1;
   // ASSJ[2] := 2;
   // ASSJ[3] := 3;
   // ASSJ[4] := 4;
   // ASSJ[5] := 5;
   // ASSJ[6] := 6;
   // ASSB[1] := 1;
   // ASSB[2] := 2;
   // ASSB[3] := 3;
   // ASSB[4] := 4;
   // ASSB[5] := 5;
   // ASSB[6] := 6;
   // PTTS[0] := 255;
   // PTTS[2] := 1;
   // PTTS[3] := 20;
   // PTTS[4] := 4;
   // PTTS[5] := 32;
   // PTTS[6] := 3;
   // NTTS[1] := 1;
   // NTTS[2] := 2;
   // NTTS[3] := 3;
   // NTTS[4] := 5;
   // NTTS[5] := 6;
   // NTTS[6] := 7;
   // SW_SQTS[1] := 1;
   // SW_SQTS[2] := 1;
   // SW_SQTS[3] := 2;
   // SW_SQTS[4] := 3;
   // SW_SQTS[5] := 3;
   // SW_SQTS[6] := 4;
   // TVX[0] := 16#1;
   // TTX[0] := 16#1;
   // TSX[0] := 16#1;
   // S00X[0] := 16#1;
   // SOFFX[0] := 16#1;
   // SONX[0] := 16#1;
   // SAX[0] := 16#1;
   // SERRX[0] := 16#1;
   // SMX[0] := 16#1;
   // S0X[0] := 16#1;
   // S1X[0] := 16#1;
   // LSTT[8] := 255;
   // ATAJ[8] := 8;
   // ATAB[8] := 8;
   // PSTT[8] := 7;
   // NSTT[8] := 23;
   // ASSJ[7] := 7;
   // ASSB[7] := 7;
   // PTTS[7] := 30;
   // NTTS[7] := 8;
   // SW_SQTS[7] := 2;
   // LSTT[9] := 255;
   // LSTT[10] := 255;
   // LSTT[11] := 255;
   // ATAJ[9] := 9;
   // ATAJ[10] := 10;
   // ATAJ[11] := 11;
   // ATAB[9] := 9;
   // ATAB[10] := 10;
   // ATAB[11] := 11;
   // PSTT[9] := 8;
   // PSTT[10] := 9;
   // PSTT[11] := 10;
   // NSTT[9] := 9;
   // NSTT[10] := 34;
   // NSTT[11] := 33;
   // ASSJ[8] := 8;
   // ASSJ[9] := 9;
   // ASSJ[10] := 10;
   // ASSB[8] := 8;
   // ASSB[9] := 9;
   // ASSB[10] := 10;
   // PTTS[8] := 23;
   // PTTS[9] := 9;
   // PTTS[10] := 36;
   // NTTS[8] := 9;
   // NTTS[9] := 10;
   // NTTS[10] := 11;
   // SW_SQTS[8] := 1;
   // SW_SQTS[9] := 1;
   // SW_SQTS[10] := 5;
   // LSTT[12] := 255;
   // LSTT[13] := 255;
   // LSTT[14] := 255;
   // LSTT[15] := 255;
   // ATAJ[12] := 12;
   // ATAJ[13] := 13;
   // ATAJ[14] := 14;
   // ATAJ[15] := 15;
   // ATAB[12] := 12;
   // ATAB[13] := 13;
   // ATAB[14] := 14;
   // ATAB[15] := 15;
   // PSTT[12] := 11;
   // PSTT[13] := 12;
   // PSTT[14] := 13;
   // PSTT[15] := 14;
   // NSTT[12] := 12;
   // NSTT[13] := 13;
   // NSTT[14] := 31;
   // NSTT[15] := 21;
   // ASSJ[11] := 11;
   // ASSJ[12] := 12;
   // ASSJ[13] := 13;
   // ASSJ[14] := 14;
   // ASSB[11] := 11;
   // ASSB[12] := 12;
   // ASSB[13] := 13;
   // ASSB[14] := 14;
   // PTTS[11] := 5;
   // PTTS[12] := 12;
   // PTTS[13] := 13;
   // PTTS[14] := 21;
   // NTTS[11] := 12;
   // NTTS[12] := 13;
   // NTTS[13] := 14;
   // NTTS[14] := 15;
   // SW_SQTS[11] := 3;
   // SW_SQTS[12] := 3;
   // SW_SQTS[13] := 3;
   // SW_SQTS[14] := 5;
   // LSTT[16] := 255;
   // ATAJ[16] := 16;
   // ATAB[16] := 16;
   // PSTT[16] := 15;
   // NSTT[16] := 22;
   // ASSJ[15] := 15;
   // ASSB[15] := 15;
   // PTTS[15] := 2;
   // NTTS[15] := 16;
   // SW_SQTS[15] := 1;
   // LSTT[17] := 255;
   // LSTT[18] := 255;
   // LSTT[19] := 255;
   // LSTT[20] := 255;
   // LSTT[21] := 255;
   // LSTT[22] := 255;
   // ATAJ[17] := 17;
   // ATAJ[18] := 18;
   // ATAJ[19] := 19;
   // ATAJ[20] := 20;
   // ATAJ[21] := 21;
   // ATAJ[22] := 22;
   // ATAB[17] := 17;
   // ATAB[18] := 18;
   // ATAB[19] := 19;
   // ATAB[20] := 20;
   // ATAB[21] := 21;
   // ATAB[22] := 22;
   // PSTT[17] := 16;
   // PSTT[18] := 17;
   // PSTT[19] := 18;
   // PSTT[20] := 19;
   // PSTT[21] := 20;
   // PSTT[22] := 21;
   // NSTT[17] := 20;
   // NSTT[18] := 28;
   // NSTT[19] := 25;
   // NSTT[20] := 3;
   // NSTT[21] := 14;
   // NSTT[22] := 32;
   // ASSJ[16] := 16;
   // ASSJ[17] := 17;
   // ASSJ[18] := 18;
   // ASSJ[19] := 19;
   // ASSJ[20] := 20;
   // ASSJ[21] := 21;
   // ASSB[16] := 16;
   // ASSB[17] := 17;
   // ASSB[18] := 18;
   // ASSB[19] := 19;
   // ASSB[20] := 20;
   // ASSB[21] := 21;
   // PTTS[16] := 35;
   // PTTS[17] := 26;
   // PTTS[18] := 24;
   // PTTS[19] := 29;
   // PTTS[20] := 17;
   // PTTS[21] := 15;
   // NTTS[16] := 17;
   // NTTS[17] := 18;
   // NTTS[18] := 19;
   // NTTS[19] := 20;
   // NTTS[20] := 21;
   // NTTS[21] := 22;
   // SW_SQTS[16] := 5;
   // SW_SQTS[17] := 2;
   // SW_SQTS[18] := 2;
   // SW_SQTS[19] := 2;
   // SW_SQTS[20] := 5;
   // SW_SQTS[21] := 5;
   // LSTT[23] := 255;
   // ATAJ[23] := 23;
   // ATAB[23] := 23;
   // PSTT[23] := 22;
   // NSTT[23] := 8;
   // ASSJ[22] := 22;
   // ASSB[22] := 22;
   // PTTS[22] := 16;
   // NTTS[22] := 23;
   // SW_SQTS[22] := 1;
   // LSTT[24] := 255;
   // LSTT[25] := 255;
   // LSTT[26] := 255;
   // LSTT[27] := 255;
   // LSTT[28] := 255;
   // LSTT[29] := 255;
   // ATAJ[24] := 24;
   // ATAJ[25] := 25;
   // ATAJ[26] := 26;
   // ATAJ[27] := 27;
   // ATAJ[28] := 28;
   // ATAJ[29] := 29;
   // ATAB[24] := 24;
   // ATAB[25] := 25;
   // ATAB[26] := 26;
   // ATAB[27] := 27;
   // ATAB[28] := 28;
   // ATAB[29] := 29;
   // PSTT[24] := 23;
   // PSTT[25] := 24;
   // PSTT[26] := 25;
   // PSTT[27] := 26;
   // PSTT[28] := 27;
   // PSTT[29] := 28;
   // NSTT[24] := 18;
   // NSTT[25] := 30;
   // NSTT[26] := 17;
   // NSTT[27] := 27;
   // NSTT[28] := 24;
   // NSTT[29] := 19;
   // ASSJ[23] := 23;
   // ASSJ[24] := 24;
   // ASSJ[25] := 25;
   // ASSJ[26] := 26;
   // ASSJ[27] := 27;
   // ASSJ[28] := 28;
   // ASSB[23] := 23;
   // ASSB[24] := 24;
   // ASSB[25] := 25;
   // ASSB[26] := 26;
   // ASSB[27] := 27;
   // ASSB[28] := 28;
   // PTTS[23] := 8;
   // PTTS[24] := 28;
   // PTTS[25] := 19;
   // PTTS[26] := 33;
   // PTTS[27] := 27;
   // PTTS[28] := 18;
   // NTTS[23] := 24;
   // NTTS[24] := 25;
   // NTTS[25] := 26;
   // NTTS[26] := 27;
   // NTTS[27] := 28;
   // NTTS[28] := 29;
   // SW_SQTS[23] := 2;
   // SW_SQTS[24] := 6;
   // SW_SQTS[25] := 2;
   // SW_SQTS[26] := 6;
   // SW_SQTS[27] := 6;
   // SW_SQTS[28] := 2;
   // LSTT[30] := 255;
   // LSTT[31] := 255;
   // ATAJ[30] := 34;
   // ATAJ[31] := 31;
   // ATAB[30] := 30;
   // ATAB[31] := 31;
   // PSTT[30] := 29;
   // PSTT[31] := 30;
   // NSTT[30] := 7;
   // NSTT[31] := 29;
   // ASSJ[29] := 29;
   // ASSB[29] := 29;
   // PTTS[29] := 31;
   // NTTS[29] := 30;
   // SW_SQTS[29] := 6;
   // LSTT[32] := 255;
   // LSTT[33] := 255;
   // LSTT[34] := 255;
   // LSTT[35] := 255;
   // LSTT[36] := 255;
   // LSTT[37] := 255;
   // LSTT[38] := 255;
   // ATAJ[32] := 32;
   // ATAJ[33] := 33;
   // ATAJ[34] := 30;
   // ATAJ[35] := 35;
   // ATAJ[36] := 38;
   // ATAJ[37] := 37;
   // ATAJ[38] := 36;
   // ATAB[32] := 32;
   // ATAB[33] := 34;
   // ATAB[34] := 33;
   // ATAB[35] := 35;
   // ATAB[36] := 37;
   // ATAB[37] := 36;
   // ATAB[38] := 38;
   // PSTT[32] := 31;
   // PSTT[33] := 32;
   // PSTT[34] := 32;
   // PSTT[35] := 33;
   // PSTT[36] := 34;
   // PSTT[37] := 34;
   // PSTT[38] := 35;
   // NSTT[32] := 5;
   // NSTT[33] := 26;
   // NSTT[34] := 7;
   // NSTT[35] := 16;
   // NSTT[36] := 10;
   // NSTT[37] := 35;
   // NSTT[38] := 10;
   // ASSJ[30] := 30;
   // ASSJ[31] := 31;
   // ASSJ[32] := 32;
   // ASSJ[33] := 33;
   // ASSJ[34] := 34;
   // ASSJ[35] := 35;
   // ASSB[30] := 30;
   // ASSB[31] := 31;
   // ASSB[32] := 32;
   // ASSB[33] := 33;
   // ASSB[34] := 34;
   // ASSB[35] := 35;
   // PTTS[30] := 25;
   // PTTS[31] := 14;
   // PTTS[32] := 22;
   // PTTS[33] := 11;
   // PTTS[34] := 10;
   // PTTS[35] := 37;
   // NTTS[30] := 31;
   // NTTS[31] := 32;
   // NTTS[32] := 33;
   // NTTS[33] := 35;
   // NTTS[34] := 36;
   // NTTS[35] := 38;
   // SW_SQTS[30] := 6;
   // SW_SQTS[31] := 3;
   // SW_SQTS[32] := 5;
   // SW_SQTS[33] := 5;
   // SW_SQTS[34] := 1;
   // SW_SQTS[35] := 7;
BEGIN
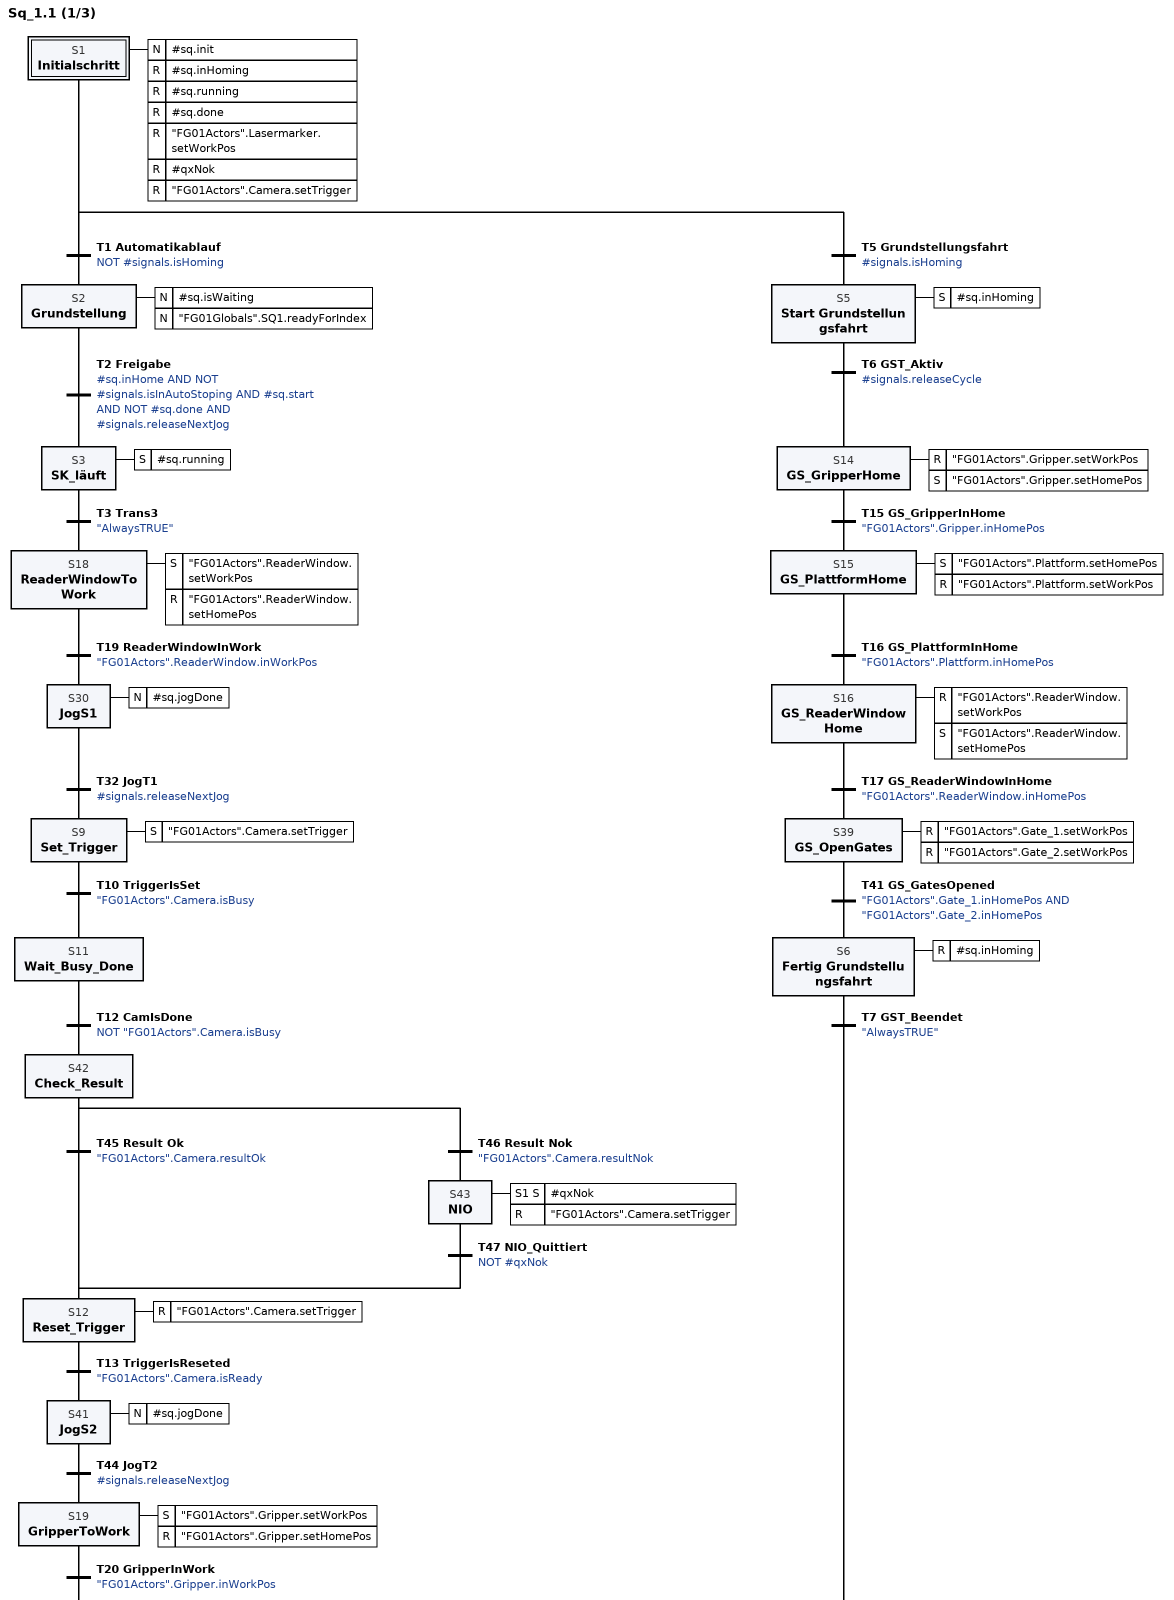
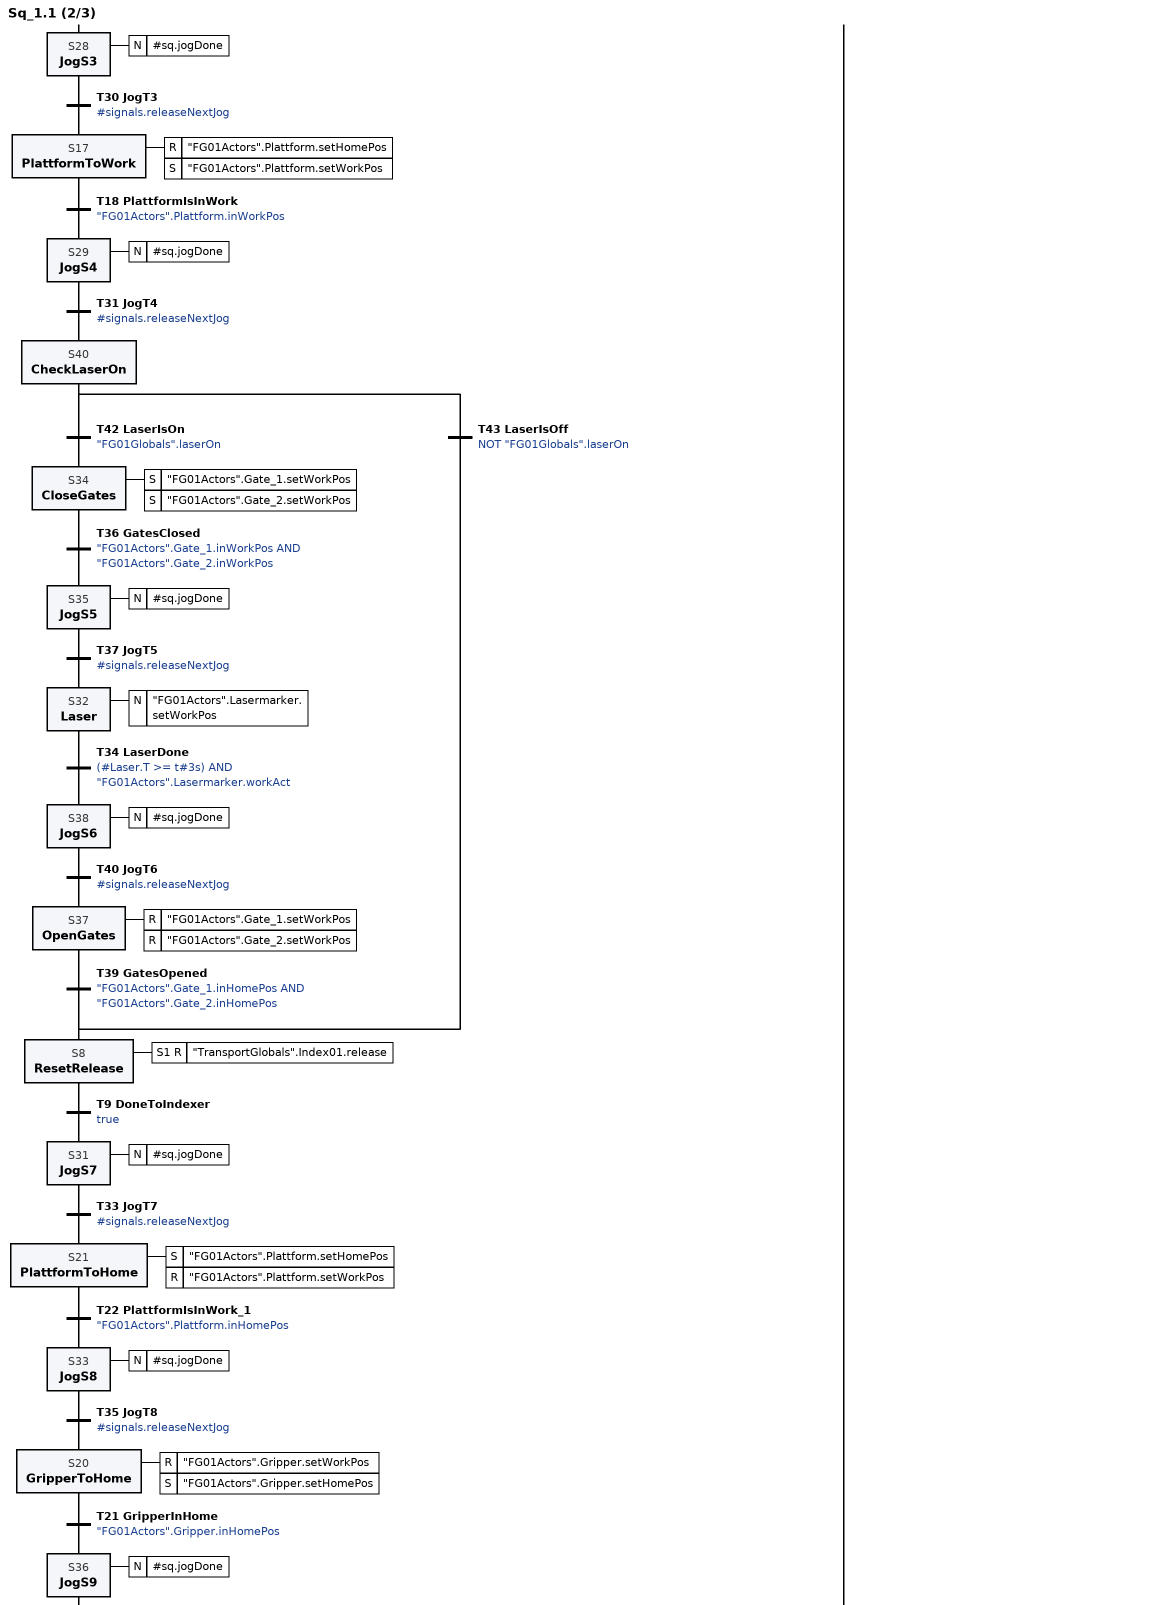
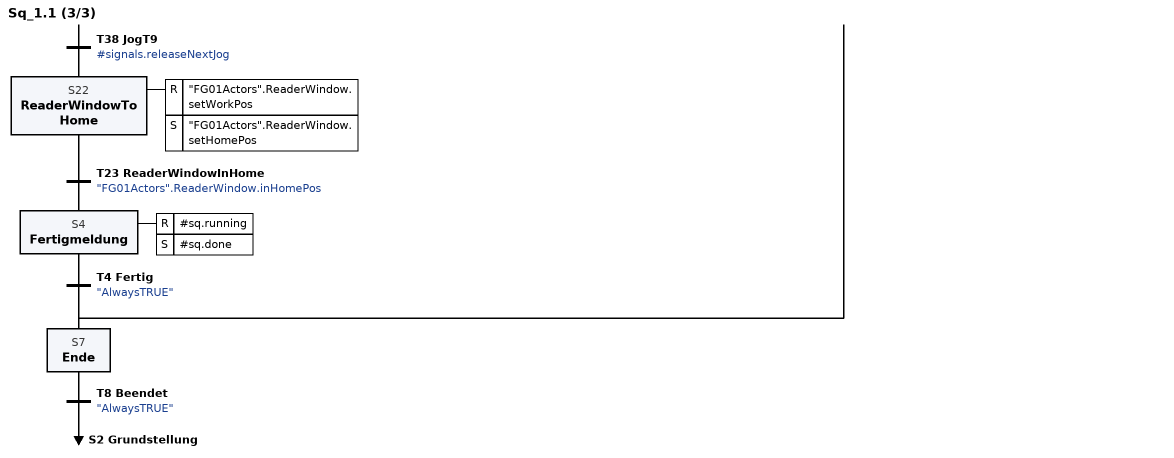
   // permanent pre-instructions
   NETWORK 1
   TITLE = Schrittkette verfügbar / Sequence available
      #sq.exists := true;
   NETWORK 2
   TITLE = Schrittkette in Grundstellung (Erweitern) / Sequence in home position (extend)
      #sq.inHome := #Grundstellung.X AND "FG01Actors".Gripper.inHomePos AND "FG01Actors".Plattform.inHomePos AND "FG01Actors".ReaderWindow.inHomePos AND "FG01Actors".Camera.isReady AND "FG01Actors".Gate_1.inHomePos AND "FG01Actors".Gate_2.inHomePos;
   NETWORK 3
   TITLE = Startbedingung (Erweitern) / Start condition (extend)
      #txStartCondition := "TransportGlobals".Index01.release;
   NETWORK 4
   TITLE = Schrittkette starten / Start sequence
      #sq.start := #sq.inHome AND NOT #sq.running AND #signals.releaseCycle AND NOT #signals.isHoming AND #txStartCondition;
      IF #sq.start THEN #sq.done := FALSE; END_IF;
   NETWORK 5
   TITLE = ReleaseCycle-Zeitgeber / ReleaseCycle timer
      // ENO of a box is taken as its EN; it also drops when the box reports an error
      #_w1 := #ERR_FLT AND #ACK_EF;
      #_w2 := #_w1 AND NOT #sstReleaseCycle.ErrorAck;   // rising edge
      #sstReleaseCycle.ErrorAck := #_w1;
      IF (#S_NO <> #sstReleaseCycle.No_LastCycle) OR #_w2 THEN
          #sstReleaseCycle.T := T#0MS;
          #sstReleaseCycle.TckPrev := #sstReleaseCycle.Tck;
          #sstReleaseCycle.No_LastCycle := #S_NO;
      END_IF;
      #sstReleaseCycle.Tck := TIME_TCK();
      #tdTckDiff := #sstReleaseCycle.Tck - #sstReleaseCycle.TckPrev;
      #sstReleaseCycle.TckPrev := #sstReleaseCycle.Tck;
      IF (0 <= #tdTckDiff) AND (#tdTckDiff <= 1000) AND #signals.releaseCycle THEN
          #sstReleaseCycle.T := #sstReleaseCycle.T + #tdTckDiff;
      END_IF;

